C05437=1065.697,216.164,-85.426,173.240,30.452,155.567
C05438=1065.691,215.915,-85.400,173.238,30.449,155.567
C05439=1065.685,215.666,-85.375,173.236,30.444,155.566
C05440=1065.680,215.418,-85.348,173.234,30.440,155.565
C05441=1065.673,215.169,-85.323,173.232,30.436,155.564
C05442=1065.668,214.920,-85.297,173.230,30.432,155.564
C05443=1065.662,214.672,-85.272,173.228,30.428,155.563
C05444=1065.655,214.423,-85.246,173.225,30.424,155.562
C05445=1065.650,214.175,-85.220,173.224,30.420,155.561
C05446=1065.643,213.926,-85.194,173.222,30.416,155.561
C05447=1065.638,213.677,-85.168,173.219,30.411,155.560
C05448=1065.632,213.428,-85.143,173.218,30.408,155.559
C05449=1065.625,213.180,-85.117,173.216,30.403,155.559
C05450=1065.620,212.931,-85.091,173.214,30.399,155.558
C05451=1065.614,212.682,-85.066,173.212,30.395,155.557
C05452=1065.608,212.435,-85.041,173.210,30.391,155.556
C05453=1065.603,212.186,-85.015,173.208,30.387,155.556
C05454=1065.596,211.937,-84.989,173.206,30.383,155.555
C05455=1065.590,211.688,-84.964,173.204,30.379,155.554
C05456=1065.585,211.439,-84.938,173.202,30.375,155.554
C05457=1065.578,211.191,-84.913,173.200,30.371,155.553
C05458=1065.572,210.942,-84.887,173.198,30.367,155.552
C05459=1065.566,210.693,-84.862,173.196,30.363,155.552
C05460=1065.560,210.445,-84.837,173.194,30.359,155.551
C05461=1065.554,210.196,-84.811,173.192,30.355,155.550
C05462=1065.549,209.948,-84.786,173.190,30.350,155.549
C05463=1065.543,209.699,-84.761,173.188,30.347,155.549
C05464=1065.536,209.450,-84.735,173.186,30.342,155.548
C05465=1065.530,209.202,-84.710,173.184,30.338,155.547
C05466=1065.525,208.982,-84.687,173.182,30.335,155.547
C05467=1065.519,208.761,-84.665,173.180,30.331,155.546
C05468=1065.514,208.541,-84.642,173.179,30.327,155.545
C05469=1065.510,208.320,-84.619,173.177,30.324,155.545
C05470=1065.504,208.100,-84.597,173.175,30.320,155.544
C05471=1065.498,207.879,-84.575,173.174,30.316,155.543
C05472=1065.493,207.659,-84.553,173.172,30.313,155.543
C05473=1065.488,207.439,-84.531,173.170,30.309,155.542
C05474=1065.464,206.392,-84.427,173.012,30.231,155.537
C05475=1065.457,206.144,-84.402,173.011,30.228,155.536
C05476=1065.452,205.895,-84.378,173.008,30.225,155.536
C05477=1065.445,205.646,-84.354,173.006,30.221,155.535
C05478=1065.440,205.398,-84.329,173.004,30.219,155.535
C05479=1065.434,205.148,-84.305,173.001,30.215,155.534
C05480=1065.429,204.900,-84.280,172.999,30.212,155.534
C05481=1065.423,204.651,-84.255,172.997,30.209,155.533
C05482=1065.417,204.402,-84.231,172.995,30.205,155.533
C05483=1065.411,204.154,-84.207,172.992,30.202,155.532
C05484=1065.406,203.905,-84.183,172.990,30.199,155.532
C05485=1065.400,203.656,-84.158,172.988,30.196,155.531
C05486=1065.394,203.407,-84.134,172.986,30.193,155.531
C05487=1065.388,203.159,-84.110,172.983,30.189,155.530
C05488=1065.383,202.910,-84.086,172.982,30.186,155.530
C05489=1065.377,202.661,-84.060,172.979,30.183,155.529
C05490=1065.371,202.413,-84.036,172.977,30.180,155.529
C05491=1065.366,202.164,-84.011,172.975,30.177,155.528
C05492=1065.360,201.915,-83.988,172.973,30.174,155.528
C05493=1065.354,201.666,-83.963,172.970,30.171,155.527
C05494=1065.348,201.418,-83.940,172.969,30.167,155.527
C05495=1065.342,201.169,-83.915,172.966,30.165,155.526
C05496=1065.336,200.920,-83.891,172.964,30.161,155.526
C05497=1065.330,200.672,-83.867,172.961,30.158,155.525
C05498=1065.324,200.422,-83.844,172.960,30.155,155.525
C05499=1065.319,200.173,-83.819,172.957,30.152,155.524
C05500=1065.312,199.924,-83.795,172.955,30.149,155.524
C05501=1065.307,199.676,-83.771,172.953,30.146,155.523
C05502=1065.301,199.428,-83.747,172.951,30.143,155.523
C05503=1065.295,199.178,-83.723,172.948,30.140,155.522
C05504=1065.289,198.930,-83.699,172.947,30.137,155.522
C05505=1065.284,198.681,-83.675,172.944,30.133,155.521
C05506=1065.277,198.432,-83.651,172.942,30.131,155.521
C05507=1065.272,198.183,-83.627,172.939,30.127,155.520
C05508=1065.265,197.934,-83.603,172.938,30.125,155.520
C05509=1065.260,197.686,-83.579,172.935,30.121,155.519
C05510=1065.254,197.437,-83.555,172.933,30.118,155.519
C05511=1065.248,197.188,-83.531,172.932,30.115,155.519
C05512=1065.242,196.940,-83.507,172.929,30.112,155.518
C05513=1065.237,196.691,-83.484,172.927,30.109,155.518
C05514=1065.230,196.442,-83.460,172.925,30.106,155.517
C05515=1065.225,196.193,-83.435,172.923,30.103,155.517
C05516=1065.219,195.945,-83.412,172.920,30.100,155.516
C05517=1065.213,195.696,-83.389,172.919,30.097,155.516
C05518=1065.207,195.447,-83.364,172.916,30.094,155.515
C05519=1065.201,195.198,-83.340,172.914,30.090,155.515
C05520=1065.196,194.950,-83.316,172.911,30.087,155.514
C05521=1065.190,194.700,-83.293,172.910,30.084,155.514
C05522=1065.184,194.452,-83.269,172.908,30.081,155.513
C05523=1065.178,194.203,-83.245,172.905,30.078,155.513
C05524=1065.173,193.954,-83.221,172.904,30.075,155.512
C05525=1065.167,193.705,-83.197,172.901,30.072,155.512
C05526=1065.161,193.457,-83.174,172.899,30.069,155.511
C05527=1065.156,193.208,-83.150,172.897,30.066,155.511
C05528=1065.150,192.959,-83.127,172.895,30.063,155.510
C05529=1065.144,192.709,-83.103,172.893,30.060,155.510
C05530=1065.138,192.461,-83.079,172.891,30.056,155.509
C05531=1065.132,192.213,-83.055,172.889,30.054,155.509
C05532=1065.127,191.964,-83.032,172.886,30.050,155.508
C05533=1065.121,191.715,-83.008,172.884,30.048,155.508
C05534=1065.115,191.465,-82.984,172.883,30.044,155.507
C05535=1065.108,191.183,-82.957,172.880,30.041,155.507
C05536=1065.102,190.900,-82.930,172.877,30.038,155.506
C05537=1065.096,190.617,-82.904,172.875,30.034,155.506
C05538=1065.090,190.334,-82.877,172.873,30.030,155.505
C05539=1065.084,190.086,-82.853,172.870,30.027,155.505
C05540=1065.078,189.837,-82.830,172.869,30.024,155.504
C05541=1065.073,189.588,-82.806,172.866,30.021,155.504
C05542=1065.067,189.340,-82.783,172.864,30.018,155.503
C05543=1065.061,189.091,-82.759,172.863,30.015,155.503
C05544=1065.055,188.841,-82.735,172.860,30.012,155.503
C05545=1065.049,188.592,-82.712,172.858,30.009,155.502
C05546=1065.044,188.344,-82.688,172.857,30.006,155.502
C05547=1065.038,188.095,-82.665,172.854,30.003,155.501
C05548=1065.032,187.847,-82.642,172.852,30.000,155.501
C05549=1065.027,187.598,-82.618,172.850,29.997,155.500
C05550=1065.022,187.349,-82.595,172.848,29.993,155.500
C05551=1065.016,187.100,-82.571,172.846,29.991,155.499
C05552=1065.011,186.851,-82.548,172.844,29.987,155.499
C05553=1065.005,186.603,-82.524,172.842,29.985,155.498
C05554=1064.998,186.353,-82.501,172.840,29.981,155.498
C05555=1064.993,186.104,-82.477,172.837,29.978,155.497
C05556=1064.987,185.856,-82.454,172.836,29.975,155.497
C05557=1064.981,185.607,-82.431,172.834,29.972,155.496
C05558=1064.976,185.358,-82.407,172.831,29.969,155.496
C05559=1064.971,185.109,-82.384,172.830,29.966,155.495
C05560=1064.965,184.861,-82.361,172.828,29.963,155.495
C05561=1064.960,184.611,-82.337,172.825,29.960,155.494
C05562=1064.954,184.362,-82.314,172.824,29.957,155.494
C05563=1064.948,184.113,-82.291,172.822,29.954,155.493
C05564=1064.942,183.865,-82.269,172.819,29.951,155.493
C05565=1064.935,183.616,-82.245,172.818,29.949,155.493
C05566=1064.929,183.367,-82.222,172.815,29.945,155.492
C05567=1064.924,183.118,-82.199,172.813,29.942,155.492
C05568=1064.918,182.869,-82.176,172.811,29.940,155.491
C05569=1064.912,182.620,-82.153,172.809,29.937,155.491
C05570=1064.906,182.371,-82.130,172.807,29.934,155.490
C05571=1064.900,182.123,-82.106,172.805,29.931,155.490
C05572=1064.893,181.874,-82.084,172.803,29.928,155.490
C05573=1064.888,181.625,-82.061,172.801,29.925,155.489
C05574=1064.882,181.376,-82.038,172.799,29.922,155.489
C05575=1064.876,181.127,-82.015,172.797,29.919,155.488
C05576=1064.870,180.878,-81.992,172.795,29.916,155.488
C05577=1064.865,180.629,-81.969,172.793,29.914,155.487
C05578=1064.859,180.381,-81.946,172.790,29.911,155.487
C05579=1064.853,180.132,-81.924,172.789,29.908,155.486
C05580=1064.847,179.883,-81.901,172.787,29.905,155.486
C05581=1064.841,179.634,-81.878,172.784,29.902,155.486
C05582=1064.835,179.385,-81.855,172.783,29.899,155.485
C05583=1064.830,179.136,-81.832,172.781,29.896,155.485
C05584=1064.824,178.887,-81.809,172.778,29.893,155.484
C05585=1064.817,178.639,-81.787,172.777,29.890,155.484
C05586=1064.812,178.390,-81.764,172.775,29.887,155.483
C05587=1064.805,178.140,-81.740,172.772,29.884,155.483
C05588=1064.800,177.891,-81.717,172.771,29.882,155.482
C05589=1064.794,177.643,-81.694,172.769,29.879,155.482
C05590=1064.788,177.394,-81.671,172.767,29.876,155.482
C05591=1064.782,177.145,-81.649,172.764,29.873,155.481
C05592=1064.776,176.896,-81.626,172.763,29.870,155.481
C05593=1064.770,176.647,-81.603,172.761,29.867,155.480
C05594=1064.765,176.398,-81.581,172.758,29.864,155.480
C05595=1064.759,176.149,-81.558,172.757,29.861,155.479
C05596=1064.753,175.901,-81.536,172.755,29.858,155.479
C05597=1064.747,175.652,-81.513,172.753,29.855,155.478
C05598=1064.742,175.403,-81.490,172.751,29.853,155.478
C05599=1064.735,175.120,-81.464,172.749,29.849,155.478
C05600=1064.729,174.836,-81.439,172.746,29.846,155.477
C05601=1064.722,174.553,-81.413,172.744,29.842,155.477
C05602=1064.716,174.270,-81.387,172.742,29.839,155.476
C05603=1064.709,174.022,-81.364,172.740,29.837,155.476
C05604=1064.704,173.772,-81.342,172.738,29.834,155.475
C05605=1064.698,173.523,-81.319,172.736,29.830,155.475
C05606=1064.692,173.274,-81.296,172.734,29.828,155.474
C05607=1064.686,173.026,-81.274,172.733,29.825,155.474
C05608=1064.680,172.776,-81.252,172.730,29.822,155.473
C05609=1064.675,172.527,-81.229,172.728,29.819,155.473
C05610=1064.669,172.278,-81.206,172.727,29.816,155.472
C05611=1064.662,172.030,-81.183,172.725,29.813,155.472
C05612=1064.658,171.781,-81.162,172.722,29.810,155.472
C05613=1064.652,171.532,-81.139,172.720,29.807,155.471
C05614=1064.646,171.283,-81.116,172.719,29.805,155.471
C05615=1064.640,171.034,-81.094,172.717,29.802,155.470
C05616=1064.634,170.785,-81.071,172.714,29.799,155.470
C05617=1064.629,170.536,-81.048,172.713,29.796,155.469
C05618=1064.623,170.287,-81.026,172.711,29.793,155.469
C05619=1064.617,170.039,-81.004,172.709,29.790,155.468
C05620=1064.612,169.790,-80.981,172.707,29.787,155.468
C05621=1064.606,169.540,-80.959,172.705,29.784,155.468
C05622=1064.600,169.292,-80.936,172.703,29.781,155.467
C05623=1064.594,169.042,-80.914,172.702,29.779,155.467
C05624=1064.589,168.794,-80.892,172.699,29.775,155.466
C05625=1064.583,168.545,-80.869,172.697,29.772,155.466
C05626=1064.577,168.296,-80.847,172.696,29.770,155.465
C05627=1064.571,168.047,-80.824,172.694,29.767,155.465
C05628=1064.566,167.798,-80.802,172.692,29.764,155.464
C05629=1064.560,167.550,-80.780,172.690,29.761,155.464
C05630=1064.555,167.300,-80.758,172.688,29.758,155.464
C05631=1064.549,167.051,-80.735,172.686,29.755,155.463
C05632=1064.543,166.802,-80.713,172.684,29.752,155.463
C05633=1064.538,166.554,-80.691,172.682,29.749,155.462
C05634=1064.532,166.304,-80.668,172.680,29.746,155.462
C05635=1064.527,166.055,-80.645,172.678,29.744,155.461
C05636=1064.520,165.806,-80.624,172.677,29.740,155.461
C05637=1064.515,165.558,-80.601,172.675,29.738,155.460
C05638=1064.510,165.308,-80.579,172.672,29.735,155.460
C05639=1064.503,165.060,-80.557,172.671,29.731,155.459
C05640=1064.498,164.810,-80.534,172.669,29.729,155.459
C05641=1064.493,164.562,-80.512,172.667,29.726,155.459
C05642=1064.487,164.313,-80.490,172.666,29.723,155.458
C05643=1064.481,164.063,-80.468,172.664,29.720,155.458
C05644=1064.476,163.815,-80.445,172.661,29.717,155.457
C05645=1064.470,163.566,-80.424,172.660,29.714,155.457
C05646=1064.465,163.317,-80.401,172.658,29.711,155.456
C05647=1064.459,163.068,-80.379,172.656,29.709,155.456
C05648=1064.453,162.819,-80.357,172.655,29.705,155.455
C05649=1064.448,162.570,-80.335,172.652,29.702,155.455
C05650=1064.442,162.322,-80.313,172.650,29.699,155.455
C05651=1064.437,162.072,-80.291,172.649,29.697,155.454
C05652=1064.431,161.823,-80.269,172.647,29.694,155.454
C05653=1064.425,161.575,-80.247,172.645,29.691,155.453
C05654=1064.420,161.325,-80.224,172.644,29.688,155.453
C05655=1064.414,161.076,-80.202,172.641,29.685,155.452
C05656=1064.409,160.827,-80.181,172.639,29.682,155.452
C05657=1064.402,160.579,-80.158,172.638,29.679,155.451
C05658=1064.396,160.329,-80.137,172.636,29.676,155.451
C05659=1064.391,160.081,-80.115,172.634,29.674,155.451
C05660=1064.385,159.831,-80.093,172.632,29.671,155.450
C05661=1064.379,159.583,-80.071,172.630,29.668,155.450
C05662=1064.373,159.333,-80.049,172.628,29.665,155.449
C05663=1064.366,159.050,-80.024,172.626,29.662,155.449
C05664=1064.361,158.766,-80.000,172.624,29.659,155.448
C05665=1064.354,158.483,-79.975,172.622,29.655,155.448
C05666=1064.347,158.199,-79.950,172.620,29.653,155.447
C05667=1064.341,157.950,-79.928,172.618,29.649,155.447
C05668=1064.335,157.701,-79.906,172.616,29.647,155.447
C05669=1064.330,157.452,-79.885,172.615,29.644,155.446
C05670=1064.324,157.203,-79.862,172.613,29.641,155.446
C05671=1064.318,156.954,-79.841,172.611,29.638,155.445
C05672=1064.312,156.706,-79.819,172.608,29.636,155.445
C05673=1064.306,156.456,-79.798,172.607,29.632,155.444
C05674=1064.301,156.207,-79.776,172.605,29.630,155.444
C05675=1064.295,155.958,-79.754,172.603,29.627,155.444
C05676=1064.289,155.709,-79.733,172.602,29.624,155.443
C05677=1064.283,155.461,-79.711,172.600,29.622,155.443
C05678=1064.278,155.211,-79.689,172.598,29.618,155.442
C05679=1064.272,154.962,-79.667,172.597,29.616,155.442
C05680=1064.266,154.713,-79.646,172.594,29.613,155.441
C05681=1064.260,154.464,-79.625,172.592,29.610,155.441
C05682=1064.254,154.215,-79.603,172.591,29.607,155.441
C05683=1064.248,153.967,-79.582,172.589,29.605,155.440
C05684=1064.243,153.717,-79.559,172.587,29.602,155.440
C05685=1064.237,153.469,-79.538,172.586,29.599,155.439
C05686=1064.231,153.219,-79.517,172.584,29.596,155.439
C05687=1064.225,152.970,-79.495,172.581,29.593,155.438
C05688=1064.219,152.722,-79.474,172.580,29.590,155.438
C05689=1064.213,152.472,-79.452,172.578,29.588,155.438
C05690=1064.208,152.224,-79.431,172.576,29.585,155.437
C05691=1064.203,151.974,-79.409,172.575,29.582,155.437
C05692=1064.197,151.725,-79.388,172.573,29.580,155.436
C05693=1064.191,151.476,-79.366,172.571,29.576,155.436
C05694=1064.185,151.227,-79.345,172.570,29.574,155.435
C05695=1064.179,150.978,-79.323,172.568,29.571,155.435
C05696=1064.173,150.729,-79.302,172.565,29.568,155.435
C05697=1064.167,150.481,-79.280,172.563,29.565,155.434
C05698=1064.162,150.231,-79.260,172.562,29.563,155.434
C05699=1064.156,149.982,-79.238,172.560,29.560,155.433
C05700=1064.150,149.733,-79.217,172.558,29.557,155.433
C05701=1064.144,149.485,-79.195,172.557,29.554,155.432
C05702=1064.139,149.235,-79.173,172.555,29.551,155.432
C05703=1064.134,148.986,-79.153,172.553,29.548,155.432
C05704=1064.127,148.737,-79.131,172.552,29.546,155.431
C05705=1064.121,148.488,-79.109,172.550,29.543,155.431
C05706=1064.116,148.239,-79.088,172.547,29.540,155.430
C05707=1064.110,147.989,-79.067,172.546,29.537,155.430
C05708=1064.104,147.741,-79.046,172.544,29.534,155.430
C05709=1064.098,147.491,-79.024,172.542,29.531,155.429
C05710=1064.092,147.243,-79.004,172.541,29.529,155.429
C05711=1064.086,146.993,-78.983,172.539,29.526,155.428
C05712=1064.080,146.745,-78.961,172.537,29.523,155.428
C05713=1064.074,146.496,-78.940,172.536,29.521,155.427
C05714=1064.069,146.247,-78.919,172.534,29.518,155.427
C05715=1064.063,145.997,-78.898,172.532,29.515,155.427
C05716=1064.057,145.749,-78.876,172.531,29.513,155.426
C05717=1064.051,145.499,-78.855,172.528,29.510,155.426
C05718=1064.046,145.251,-78.834,172.526,29.507,155.425
C05719=1064.039,145.002,-78.813,172.525,29.504,155.425
C05720=1064.034,144.753,-78.793,172.523,29.502,155.425
C05721=1064.028,144.503,-78.771,172.521,29.498,155.424
C05722=1064.022,144.254,-78.750,172.520,29.496,155.424
C05723=1064.016,144.005,-78.729,172.518,29.493,155.423
C05724=1064.011,143.757,-78.707,172.516,29.490,155.423
C05725=1064.005,143.507,-78.687,172.515,29.487,155.422
C05726=1063.998,143.259,-78.666,172.513,29.485,155.422
C05727=1063.990,142.870,-78.633,172.510,29.481,155.421
C05728=1063.981,142.481,-78.600,172.507,29.476,155.421
C05729=1063.972,142.093,-78.567,172.504,29.472,155.420
C05730=1063.963,141.704,-78.535,172.502,29.467,155.419
C05731=1063.957,141.454,-78.514,172.500,29.464,155.419
C05732=1063.951,141.206,-78.493,172.499,29.462,155.419
C05733=1063.946,140.956,-78.472,172.497,29.459,155.418
C05734=1063.940,140.707,-78.451,172.495,29.456,155.418
C05735=1063.931,140.314,-78.418,172.492,29.452,155.417
C05736=1063.921,139.920,-78.385,172.489,29.447,155.416
C05737=1063.912,139.528,-78.352,172.487,29.443,155.416
C05738=1063.903,139.134,-78.319,172.484,29.439,155.415
C05739=1063.898,138.885,-78.298,172.483,29.436,155.415
C05740=1063.891,138.636,-78.278,172.481,29.433,155.414
C05741=1063.886,138.387,-78.257,172.479,29.431,155.414
C05742=1063.880,138.137,-78.236,172.478,29.428,155.413
C05743=1063.874,137.889,-78.216,172.476,29.425,155.413
C05744=1063.868,137.639,-78.195,172.474,29.422,155.413
C05745=1063.862,137.390,-78.173,172.472,29.419,155.412
C05746=1063.856,137.141,-78.153,172.470,29.417,155.412
C05747=1063.851,136.892,-78.133,172.468,29.414,155.411
C05748=1063.844,136.643,-78.112,172.467,29.411,155.411
C05749=1063.839,136.394,-78.091,172.465,29.409,155.411
C05750=1063.833,136.144,-78.070,172.463,29.406,155.410
C05751=1063.827,135.896,-78.050,172.462,29.403,155.410
C05752=1063.821,135.647,-78.029,172.460,29.401,155.409
C05753=1063.815,135.398,-78.009,172.458,29.398,155.409
C05754=1063.809,135.149,-77.988,172.456,29.395,155.409
C05755=1063.804,134.900,-77.967,172.455,29.392,155.408
C05756=1063.797,134.650,-77.947,172.453,29.390,155.408
C05757=1063.792,134.401,-77.926,172.452,29.386,155.407
C05758=1063.786,134.153,-77.906,172.450,29.384,155.407
C05759=1063.780,133.903,-77.885,172.448,29.381,155.406
C05760=1063.775,133.654,-77.864,172.447,29.378,155.406
C05761=1063.769,133.405,-77.844,172.445,29.375,155.406
C05762=1063.763,133.156,-77.823,172.443,29.373,155.405
C05763=1063.757,132.907,-77.803,172.441,29.370,155.405
C05764=1063.752,132.658,-77.783,172.440,29.367,155.404
C05765=1063.746,132.409,-77.761,172.438,29.365,155.404
C05766=1063.739,132.160,-77.741,172.436,29.362,155.404
C05767=1063.734,131.911,-77.720,172.435,29.359,155.403
C05768=1063.728,131.662,-77.700,172.433,29.356,155.403
C05769=1063.722,131.412,-77.680,172.431,29.354,155.402
C05770=1063.716,131.163,-77.660,172.430,29.351,155.402
C05771=1063.710,130.914,-77.640,172.428,29.348,155.402
C05772=1063.704,130.665,-77.619,172.426,29.346,155.401
C05773=1063.698,130.416,-77.599,172.425,29.343,155.401
C05774=1063.692,130.167,-77.579,172.423,29.340,155.400
C05775=1063.686,129.918,-77.559,172.421,29.337,155.400
C05776=1063.681,129.668,-77.538,172.420,29.335,155.400
C05777=1063.675,129.419,-77.518,172.418,29.332,155.399
C05778=1063.668,129.171,-77.497,172.416,29.329,155.399
C05779=1063.662,128.921,-77.476,172.415,29.327,155.398
C05780=1063.656,128.673,-77.456,172.413,29.324,155.398
C05781=1063.650,128.424,-77.436,172.411,29.322,155.398
C05782=1063.645,128.174,-77.417,172.410,29.319,155.397
C05783=1063.639,127.924,-77.396,172.408,29.316,155.397
C05784=1063.633,127.676,-77.376,172.406,29.314,155.396
C05785=1063.627,127.427,-77.356,172.405,29.311,155.396
C05786=1063.621,127.177,-77.335,172.403,29.308,155.396
C05787=1063.614,126.894,-77.312,172.401,29.305,155.395
C05788=1063.607,126.610,-77.290,172.399,29.302,155.395
C05789=1063.601,126.326,-77.267,172.397,29.299,155.394
C05790=1063.594,126.042,-77.243,172.396,29.296,155.394
C05791=1063.589,125.792,-77.224,172.394,29.293,155.393
C05792=1063.583,125.543,-77.204,172.392,29.290,155.393
C05793=1063.576,125.294,-77.183,172.391,29.288,155.393
C05794=1063.570,125.045,-77.163,172.389,29.285,155.392
C05795=1063.565,124.796,-77.143,172.387,29.282,155.392
C05796=1063.559,124.547,-77.123,172.386,29.279,155.391
C05797=1063.553,124.298,-77.103,172.384,29.277,155.391
C05798=1063.546,124.049,-77.082,172.382,29.274,155.391
C05799=1063.541,123.799,-77.063,172.381,29.271,155.390
C05800=1063.535,123.550,-77.043,172.379,29.269,155.390
C05801=1063.529,123.301,-77.023,172.377,29.266,155.389
C05802=1063.523,123.053,-77.003,172.376,29.263,155.389
C05803=1063.518,122.803,-76.982,172.374,29.260,155.388
C05804=1063.512,122.553,-76.963,172.372,29.258,155.388
C05805=1063.506,122.304,-76.943,172.371,29.255,155.388
C05806=1063.500,122.056,-76.923,172.369,29.252,155.387
C05807=1063.495,121.807,-76.902,172.367,29.250,155.387
C05808=1063.489,121.557,-76.883,172.366,29.247,155.386
C05809=1063.483,121.308,-76.863,172.365,29.244,155.386
C05810=1063.476,121.059,-76.843,172.363,29.242,155.386
C05811=1063.470,120.810,-76.823,172.362,29.239,155.385
C05812=1063.465,120.560,-76.803,172.360,29.236,155.385
C05813=1063.459,120.311,-76.783,172.358,29.233,155.384
C05814=1063.453,120.063,-76.763,172.357,29.231,155.384
C05815=1063.447,119.814,-76.743,172.355,29.228,155.384
C05816=1063.443,119.564,-76.723,172.353,29.225,155.383
C05817=1063.437,119.315,-76.703,172.352,29.222,155.383
C05818=1063.431,119.066,-76.683,172.350,29.219,155.382
C05819=1063.425,118.817,-76.664,172.348,29.216,155.382
C05820=1063.418,118.567,-76.644,172.347,29.214,155.381
C05821=1063.413,118.318,-76.623,172.345,29.211,155.381
C05822=1063.407,118.069,-76.604,172.343,29.208,155.381
C05823=1063.401,117.820,-76.584,172.342,29.205,155.380
C05824=1063.396,117.571,-76.565,172.340,29.203,155.380
C05825=1063.390,117.322,-76.545,172.338,29.200,155.379
C05826=1063.384,117.073,-76.524,172.337,29.197,155.379
C05827=1063.379,116.823,-76.505,172.335,29.195,155.379
C05828=1063.373,116.574,-76.485,172.334,29.192,155.378
C05829=1063.367,116.325,-76.466,172.333,29.189,155.378
C05830=1063.361,116.076,-76.446,172.331,29.187,155.377
C05831=1063.355,115.827,-76.426,172.329,29.184,155.377
C05832=1063.350,115.578,-76.406,172.328,29.181,155.377
C05833=1063.344,115.329,-76.386,172.326,29.178,155.376
C05834=1063.338,115.079,-76.367,172.325,29.175,155.376
C05835=1063.332,114.831,-76.347,172.323,29.172,155.375
C05836=1063.327,114.581,-76.327,172.321,29.170,155.375
C05837=1063.321,114.332,-76.308,172.320,29.167,155.374
C05838=1063.316,114.083,-76.288,172.318,29.164,155.374
C05839=1063.309,113.834,-76.268,172.316,29.161,155.374
C05840=1063.303,113.585,-76.249,172.315,29.159,155.373
C05841=1063.297,113.336,-76.229,172.313,29.156,155.373
C05842=1063.292,113.086,-76.210,172.312,29.153,155.372
C05843=1063.286,112.838,-76.190,172.311,29.151,155.372
C05844=1063.280,112.588,-76.171,172.309,29.148,155.372
C05845=1063.274,112.339,-76.151,172.307,29.145,155.371
C05846=1063.268,112.090,-76.131,172.306,29.142,155.371
C05847=1063.263,111.841,-76.112,172.304,29.140,155.370
C05848=1063.257,111.592,-76.092,172.302,29.137,155.370
C05849=1063.251,111.342,-76.073,172.301,29.134,155.370
C05850=1063.245,111.093,-76.054,172.299,29.132,155.369
C05851=1063.238,110.808,-76.031,172.297,29.129,155.369
C05852=1063.232,110.525,-76.009,172.296,29.126,155.368
C05853=1063.224,110.240,-75.987,172.294,29.123,155.368
C05854=1063.217,109.957,-75.965,172.292,29.120,155.367
C05855=1063.212,109.707,-75.946,172.290,29.117,155.367
C05856=1063.206,109.458,-75.926,172.289,29.115,155.367
C05857=1063.200,109.209,-75.907,172.288,29.112,155.366
C05858=1063.194,108.960,-75.888,172.286,29.109,155.366
C05859=1063.188,108.710,-75.869,172.284,29.106,155.365
C05860=1063.182,108.461,-75.849,172.283,29.104,155.365
C05861=1063.176,108.212,-75.830,172.281,29.101,155.365
C05862=1063.171,107.963,-75.810,172.279,29.098,155.364
C05863=1063.164,107.714,-75.791,172.278,29.095,155.364
C05864=1063.158,107.465,-75.772,172.276,29.093,155.363
C05865=1063.152,107.215,-75.752,172.274,29.090,155.363
C05866=1063.147,106.966,-75.733,172.273,29.087,155.363
C05867=1063.140,106.717,-75.715,172.271,29.084,155.362
C05868=1063.134,106.468,-75.695,172.270,29.082,155.362
C05869=1063.129,106.218,-75.675,172.269,29.079,155.361
C05870=1063.123,105.969,-75.656,172.267,29.077,155.361
C05871=1063.117,105.720,-75.637,172.265,29.074,155.361
C05872=1063.111,105.471,-75.619,172.264,29.071,155.360
C05873=1063.105,105.222,-75.599,172.262,29.069,155.360
C05874=1063.100,104.973,-75.579,172.260,29.066,155.359
C05875=1063.094,104.723,-75.560,172.259,29.063,155.359
C05876=1063.088,104.474,-75.541,172.257,29.061,155.359
C05877=1063.082,104.225,-75.522,172.256,29.058,155.358
C05878=1063.076,103.975,-75.503,172.255,29.055,155.358
C05879=1063.070,103.727,-75.483,172.253,29.053,155.357
C05880=1063.064,103.478,-75.464,172.252,29.050,155.357
C05881=1063.058,103.228,-75.445,172.250,29.047,155.357
C05882=1063.053,102.979,-75.426,172.248,29.044,155.356
C05883=1063.047,102.730,-75.408,172.247,29.042,155.356
C05884=1063.041,102.481,-75.388,172.245,29.039,155.355
C05885=1063.035,102.231,-75.369,172.243,29.036,155.355
C05886=1063.030,101.982,-75.350,172.242,29.033,155.355
C05887=1063.023,101.733,-75.331,172.241,29.031,155.354
C05888=1063.017,101.483,-75.312,172.239,29.028,155.354
C05889=1063.012,101.235,-75.293,172.238,29.025,155.353
C05890=1063.007,100.985,-75.274,172.236,29.023,155.353
C05891=1063.000,100.736,-75.255,172.234,29.020,155.353
C05892=1062.995,100.487,-75.236,172.233,29.017,155.352
C05893=1062.988,100.238,-75.217,172.231,29.014,155.352
C05894=1062.982,99.988,-75.198,172.230,29.012,155.351
C05895=1062.976,99.739,-75.179,172.228,29.009,155.351
C05896=1062.970,99.490,-75.160,172.227,29.006,155.350
C05897=1062.964,99.240,-75.142,172.226,29.004,155.350
C05898=1062.959,98.992,-75.123,172.224,29.001,155.350
C05899=1062.952,98.743,-75.104,172.222,28.999,155.349
C05900=1062.947,98.493,-75.085,172.221,28.996,155.349
C05901=1062.940,98.244,-75.066,172.219,28.993,155.349
C05902=1062.935,97.995,-75.047,172.217,28.990,155.348
C05903=1062.928,97.745,-75.028,172.216,28.988,155.348
C05904=1062.923,97.496,-75.009,172.214,28.985,155.347
C05905=1062.917,97.248,-74.991,172.213,28.982,155.347
C05906=1062.911,96.998,-74.971,172.212,28.980,155.347
C05907=1062.905,96.748,-74.954,172.210,28.977,155.346
C05908=1062.899,96.499,-74.934,172.208,28.975,155.346
C05909=1062.893,96.250,-74.916,172.207,28.972,155.345
C05910=1062.888,96.001,-74.897,172.205,28.969,155.345
C05911=1062.881,95.752,-74.878,172.204,28.966,155.345
C05912=1062.875,95.503,-74.859,172.202,28.964,155.344
C05913=1062.869,95.254,-74.840,172.201,28.961,155.344
C05914=1062.863,95.004,-74.822,172.200,28.958,155.343
C05915=1062.857,94.719,-74.801,172.198,28.955,155.343
C05916=1062.850,94.436,-74.780,172.195,28.952,155.343
C05917=1062.843,94.152,-74.757,172.194,28.949,155.342
C05918=1062.836,93.868,-74.736,172.192,28.946,155.342
C05919=1062.830,93.618,-74.718,172.191,28.943,155.341
C05920=1062.825,93.369,-74.700,172.189,28.940,155.341
C05921=1062.819,93.120,-74.681,172.188,28.938,155.340
C05922=1062.813,92.871,-74.662,172.187,28.935,155.340
C05923=1062.807,92.621,-74.644,172.185,28.932,155.340
C05924=1062.802,92.372,-74.625,172.183,28.930,155.339
C05925=1062.795,92.123,-74.606,172.182,28.927,155.339
C05926=1062.790,91.874,-74.587,172.180,28.924,155.338
C05927=1062.784,91.625,-74.569,172.178,28.921,155.338
C05928=1062.778,91.376,-74.551,172.178,28.919,155.338
C05929=1062.772,91.126,-74.531,172.176,28.916,155.337
C05930=1062.766,90.876,-74.514,172.175,28.913,155.337
C05931=1062.761,90.628,-74.495,172.173,28.911,155.336
C05932=1062.754,90.379,-74.476,172.171,28.908,155.336
C05933=1062.748,90.129,-74.458,172.170,28.906,155.336
C05934=1062.742,89.880,-74.439,172.168,28.903,155.335
C05935=1062.736,89.631,-74.421,172.166,28.900,155.335
C05936=1062.731,89.381,-74.403,172.166,28.898,155.334
C05937=1062.724,89.132,-74.384,172.164,28.895,155.334
C05938=1062.718,88.882,-74.366,172.162,28.892,155.334
C05939=1062.712,88.634,-74.348,172.161,28.890,155.333
C05940=1062.707,88.385,-74.328,172.159,28.887,155.333
C05941=1062.700,88.135,-74.311,172.157,28.884,155.333
C05942=1062.694,87.886,-74.292,172.156,28.882,155.332
C05943=1062.688,87.637,-74.274,172.155,28.879,155.332
C05944=1062.682,87.388,-74.256,172.154,28.876,155.331
C05945=1062.676,87.138,-74.238,172.152,28.874,155.331
C05946=1062.671,86.889,-74.219,172.150,28.871,155.331
C05947=1062.664,86.640,-74.200,172.149,28.869,155.330
C05948=1062.658,86.390,-74.182,172.147,28.866,155.330
C05949=1062.652,86.141,-74.164,172.145,28.863,155.329
C05950=1062.646,85.892,-74.146,172.145,28.861,155.329
C05951=1062.641,85.643,-74.127,172.143,28.858,155.329
C05952=1062.635,85.393,-74.109,172.141,28.855,155.328
C05953=1062.629,85.144,-74.091,172.140,28.852,155.328
C05954=1062.623,84.895,-74.073,172.138,28.850,155.327
C05955=1062.616,84.646,-74.054,172.136,28.847,155.327
C05956=1062.611,84.397,-74.036,172.135,28.845,155.327
C05957=1062.605,84.147,-74.019,172.134,28.842,155.326
C05958=1062.599,83.897,-73.999,172.133,28.839,155.326
C05959=1062.593,83.648,-73.982,172.131,28.837,155.326
C05960=1062.587,83.399,-73.963,172.129,28.834,155.325
C05961=1062.581,83.150,-73.946,172.128,28.831,155.325
C05962=1062.575,82.901,-73.927,172.126,28.828,155.324
C05963=1062.569,82.651,-73.909,172.124,28.826,155.324
C05964=1062.564,82.402,-73.891,172.124,28.823,155.323
C05965=1062.558,82.153,-73.872,172.122,28.820,155.323
C05966=1062.552,81.903,-73.854,172.120,28.818,155.323
C05967=1062.546,81.655,-73.836,172.119,28.815,155.322
C05968=1062.540,81.405,-73.818,172.117,28.813,155.322
C05969=1062.534,81.156,-73.800,172.116,28.810,155.322
C05970=1062.528,80.907,-73.782,172.115,28.807,155.321
C05971=1062.522,80.658,-73.764,172.113,28.804,155.321
C05972=1062.517,80.408,-73.746,172.112,28.802,155.320
C05973=1062.510,80.159,-73.727,172.110,28.799,155.320
C05974=1062.505,79.910,-73.709,172.108,28.796,155.320
C05975=1062.499,79.660,-73.692,172.107,28.793,155.319
C05976=1062.493,79.411,-73.673,172.105,28.791,155.319
C05977=1062.487,79.162,-73.655,172.105,28.788,155.318
C05978=1062.481,78.913,-73.638,172.103,28.785,155.318
C05979=1062.474,78.629,-73.617,172.101,28.783,155.318
C05980=1062.468,78.344,-73.596,172.100,28.779,155.317
C05981=1062.461,78.059,-73.576,172.098,28.776,155.317
C05982=1062.454,77.775,-73.555,172.096,28.774,155.316
C05983=1062.448,77.526,-73.538,172.095,28.771,155.316
C05984=1062.442,77.277,-73.520,172.093,28.768,155.315
C05985=1062.436,77.029,-73.502,172.092,28.765,155.315
C05986=1062.430,76.779,-73.484,172.090,28.763,155.315
C05987=1062.424,76.530,-73.466,172.088,28.760,155.314
C05988=1062.418,76.280,-73.448,172.087,28.758,155.314
C05989=1062.412,76.030,-73.431,172.086,28.755,155.314
C05990=1062.406,75.782,-73.412,172.084,28.752,155.313
C05991=1062.400,75.532,-73.394,172.083,28.750,155.313
C05992=1062.394,75.283,-73.377,172.081,28.747,155.312
C05993=1062.388,75.033,-73.359,172.080,28.744,155.312
C05994=1062.382,74.785,-73.342,172.078,28.741,155.312
C05995=1062.376,74.535,-73.324,172.076,28.739,155.311
C05996=1062.370,74.286,-73.306,172.076,28.737,155.311
C05997=1062.364,74.036,-73.288,172.074,28.734,155.310
C05998=1062.358,73.788,-73.270,172.072,28.731,155.310
C05999=1062.352,73.538,-73.252,172.071,28.728,155.310
C06000=1062.347,73.289,-73.235,172.069,28.726,155.309
C06001=1062.341,73.039,-73.217,172.068,28.723,155.309
C06002=1062.334,72.790,-73.200,172.067,28.721,155.309
C06003=1062.328,72.541,-73.182,172.065,28.718,155.308
C06004=1062.323,72.292,-73.164,172.064,28.715,155.308
C06005=1062.317,72.042,-73.146,172.062,28.712,155.307
C06006=1062.311,71.793,-73.129,172.060,28.710,155.307
C06007=1062.305,71.543,-73.111,172.059,28.707,155.307
C06008=1062.299,71.294,-73.094,172.058,28.704,155.306
C06009=1062.293,71.045,-73.076,172.057,28.702,155.306
C06010=1062.287,70.796,-73.058,172.055,28.699,155.305
C06011=1062.281,70.546,-73.040,172.053,28.697,155.305
C06012=1062.275,70.297,-73.023,172.052,28.694,155.305
C06013=1062.269,70.047,-73.006,172.050,28.691,155.304
C06014=1062.263,69.798,-72.988,172.049,28.689,155.304
C06015=1062.257,69.549,-72.970,172.048,28.686,155.303
C06016=1062.251,69.300,-72.952,172.046,28.683,155.303
C06017=1062.245,69.050,-72.935,172.044,28.681,155.303
C06018=1062.239,68.801,-72.918,172.043,28.678,155.302
C06019=1062.233,68.551,-72.900,172.041,28.675,155.302
C06020=1062.227,68.303,-72.883,172.041,28.673,155.301
C06021=1062.221,68.054,-72.865,172.039,28.670,155.301
C06022=1062.215,67.804,-72.847,172.037,28.667,155.301
C06023=1062.210,67.555,-72.830,172.036,28.665,155.300
C06024=1062.203,67.305,-72.813,172.034,28.662,155.300
C06025=1062.197,67.056,-72.795,172.032,28.659,155.300
C06026=1062.191,66.806,-72.777,172.032,28.657,155.299
C06027=1062.185,66.557,-72.760,172.030,28.654,155.299
C06028=1062.179,66.308,-72.743,172.029,28.652,155.299
C06029=1062.173,66.059,-72.726,172.027,28.649,155.298
C06030=1062.167,65.810,-72.708,172.025,28.646,155.298
C06031=1062.161,65.559,-72.691,172.024,28.644,155.297
C06032=1062.155,65.311,-72.674,172.023,28.641,155.297
C06033=1062.149,65.061,-72.656,172.021,28.638,155.297
C06034=1062.143,64.812,-72.638,172.020,28.636,155.296
C06035=1062.137,64.563,-72.621,172.018,28.633,155.296
C06036=1062.131,64.313,-72.603,172.017,28.630,155.295
C06037=1062.125,64.064,-72.587,172.015,28.628,155.295
C06038=1062.119,63.814,-72.569,172.014,28.626,155.295
C06039=1062.113,63.566,-72.552,172.013,28.623,155.294
C06040=1062.107,63.316,-72.534,172.011,28.620,155.294
C06041=1062.101,63.067,-72.518,172.009,28.617,155.294
C06042=1062.094,62.817,-72.501,172.008,28.615,155.293
C06043=1062.088,62.533,-72.481,172.006,28.612,155.293
C06044=1062.080,62.249,-72.461,172.005,28.609,155.292
C06045=1062.073,61.964,-72.442,172.003,28.606,155.292
C06046=1062.066,61.680,-72.423,172.001,28.604,155.292
C06047=1062.060,61.431,-72.405,172.000,28.601,155.291
C06048=1062.054,61.182,-72.388,171.998,28.598,155.291
C06049=1062.048,60.933,-72.372,171.996,28.596,155.290
C06050=1062.042,60.683,-72.354,171.996,28.593,155.290
C06051=1062.036,60.434,-72.337,171.994,28.590,155.290
C06052=1062.030,60.184,-72.319,171.993,28.588,155.289
C06053=1062.024,59.935,-72.302,171.991,28.585,155.289
C06054=1062.018,59.686,-72.286,171.989,28.583,155.289
C06055=1062.012,59.436,-72.268,171.988,28.580,155.288
C06056=1062.005,59.187,-72.251,171.987,28.578,155.288
C06057=1062.000,58.937,-72.234,171.985,28.575,155.287
C06058=1061.993,58.688,-72.217,171.984,28.572,155.287
C06059=1061.987,58.439,-72.201,171.982,28.570,155.287
C06060=1061.981,58.189,-72.183,171.981,28.567,155.286
C06061=1061.975,57.940,-72.166,171.979,28.565,155.286
C06062=1061.969,57.691,-72.150,171.978,28.562,155.286
C06063=1061.963,57.441,-72.132,171.977,28.559,155.285
C06064=1061.957,57.192,-72.116,171.975,28.557,155.285
C06065=1061.951,56.943,-72.099,171.973,28.554,155.285
C06066=1061.945,56.693,-72.081,171.972,28.551,155.284
C06067=1061.939,56.444,-72.064,171.970,28.549,155.284
C06068=1061.933,56.195,-72.048,171.970,28.547,155.283
C06069=1061.927,55.945,-72.030,171.968,28.544,155.283
C06070=1061.921,55.696,-72.014,171.966,28.541,155.283
C06071=1061.914,55.447,-71.997,171.965,28.538,155.282
C06072=1061.909,55.197,-71.980,171.963,28.536,155.282
C06073=1061.902,54.948,-71.963,171.961,28.533,155.282
C06074=1061.896,54.699,-71.947,171.961,28.531,155.281
C06075=1061.891,54.449,-71.929,171.959,28.528,155.281
C06076=1061.884,54.199,-71.912,171.958,28.526,155.280
C06077=1061.878,53.951,-71.895,171.956,28.523,155.280
C06078=1061.873,53.701,-71.878,171.954,28.520,155.280
C06079=1061.866,53.452,-71.862,171.953,28.517,155.279
C06080=1061.860,53.202,-71.845,171.952,28.515,155.279
C06081=1061.854,52.953,-71.827,171.950,28.513,155.279
C06082=1061.848,52.704,-71.811,171.949,28.510,155.278
C06083=1061.843,52.455,-71.795,171.947,28.507,155.278
C06084=1061.836,52.205,-71.777,171.946,28.505,155.278
C06085=1061.830,51.955,-71.761,171.945,28.502,155.277
C06086=1061.824,51.707,-71.744,171.943,28.500,155.277
C06087=1061.819,51.457,-71.727,171.942,28.497,155.276
C06088=1061.813,51.208,-71.711,171.940,28.494,155.276
C06089=1061.806,50.958,-71.693,171.939,28.492,155.276
C06090=1061.800,50.709,-71.677,171.937,28.489,155.275
C06091=1061.795,50.459,-71.660,171.936,28.486,155.275
C06092=1061.789,50.211,-71.643,171.935,28.484,155.274
C06093=1061.783,49.961,-71.627,171.933,28.481,155.274
C06094=1061.777,49.711,-71.610,171.931,28.479,155.274
C06095=1061.771,49.462,-71.593,171.930,28.476,155.273
C06096=1061.765,49.213,-71.576,171.928,28.473,155.273
C06097=1061.759,48.963,-71.560,171.928,28.470,155.273
C06098=1061.753,48.714,-71.543,171.926,28.468,155.272
C06099=1061.747,48.464,-71.526,171.924,28.465,155.272
C06100=1061.741,48.215,-71.510,171.923,28.463,155.271
C06101=1061.735,47.966,-71.493,171.921,28.460,155.271
C06102=1061.729,47.717,-71.476,171.921,28.457,155.271
C06103=1061.723,47.467,-71.460,171.919,28.455,155.270
C06104=1061.717,47.218,-71.443,171.917,28.452,155.270
C06105=1061.712,46.968,-71.427,171.916,28.450,155.270
C06106=1061.705,46.719,-71.409,171.914,28.447,155.269
C06107=1061.699,46.435,-71.391,171.913,28.444,155.269
C06108=1061.692,46.150,-71.372,171.911,28.441,155.268
C06109=1061.685,45.865,-71.353,171.909,28.438,155.268
C06110=1061.679,45.581,-71.334,171.908,28.435,155.267
C06111=1061.673,45.332,-71.318,171.906,28.432,155.267
C06112=1061.667,45.082,-71.301,171.905,28.429,155.267
C06113=1061.661,44.833,-71.284,171.903,28.427,155.266
C06114=1061.655,44.584,-71.268,171.902,28.425,155.266
C06115=1061.649,44.334,-71.251,171.901,28.422,155.266
C06116=1061.644,44.085,-71.235,171.899,28.419,155.265
C06117=1061.638,43.835,-71.218,171.898,28.416,155.265
C06118=1061.632,43.586,-71.202,171.896,28.413,155.264
C06119=1061.626,43.336,-71.186,171.895,28.411,155.264
C06120=1061.620,43.087,-71.170,171.894,28.409,155.264
C06121=1061.613,42.838,-71.152,171.892,28.406,155.263
C06122=1061.607,42.588,-71.136,171.890,28.404,155.263
C06123=1061.601,42.339,-71.120,171.889,28.401,155.263
C06124=1061.595,42.090,-71.103,171.887,28.398,155.262
C06125=1061.589,41.840,-71.087,171.887,28.396,155.262
C06126=1061.583,41.591,-71.071,171.885,28.393,155.262
C06127=1061.577,41.342,-71.055,171.883,28.391,155.261
C06128=1061.571,41.092,-71.038,171.882,28.388,155.261
C06129=1061.565,40.843,-71.022,171.880,28.385,155.260
C06130=1061.559,40.593,-71.005,171.879,28.383,155.260
C06131=1061.553,40.343,-70.989,171.878,28.380,155.260
C06132=1061.547,40.094,-70.973,171.876,28.378,155.259
C06133=1061.541,39.845,-70.957,171.875,28.375,155.259
C06134=1061.535,39.595,-70.940,171.873,28.372,155.259
C06135=1061.529,39.346,-70.924,171.871,28.370,155.258
C06136=1061.523,39.097,-70.908,171.870,28.367,155.258
C06137=1061.517,38.847,-70.892,171.869,28.365,155.257
C06138=1061.511,38.598,-70.875,171.868,28.362,155.257
C06139=1061.505,38.349,-70.859,171.866,28.360,155.257
C06140=1061.499,38.099,-70.843,171.864,28.357,155.256
C06141=1061.493,37.850,-70.827,171.863,28.354,155.256
C06142=1061.487,37.601,-70.810,171.861,28.352,155.256
C06143=1061.481,37.351,-70.794,171.861,28.349,155.255
C06144=1061.475,37.102,-70.778,171.859,28.347,155.255
C06145=1061.469,36.852,-70.763,171.857,28.344,155.255
C06146=1061.463,36.602,-70.746,171.856,28.342,155.254
C06147=1061.457,36.353,-70.730,171.854,28.339,155.254
C06148=1061.451,36.104,-70.714,171.853,28.336,155.254
C06149=1061.445,35.854,-70.698,171.852,28.335,155.253
C06150=1061.438,35.605,-70.682,171.850,28.332,155.253
C06151=1061.432,35.356,-70.666,171.849,28.329,155.253
C06152=1061.426,35.106,-70.650,171.847,28.327,155.252
C06153=1061.420,34.857,-70.634,171.845,28.324,155.252
C06154=1061.414,34.607,-70.618,171.844,28.321,155.251
C06155=1061.408,34.358,-70.602,171.843,28.319,155.251
C06156=1061.402,34.109,-70.586,171.842,28.316,155.251
C06157=1061.396,33.859,-70.569,171.840,28.314,155.250
C06158=1061.390,33.609,-70.554,171.838,28.311,155.250
C06159=1061.384,33.360,-70.538,171.837,28.308,155.250
C06160=1061.378,33.111,-70.522,171.835,28.306,155.249
C06161=1061.372,32.862,-70.506,171.834,28.304,155.249
C06162=1061.366,32.612,-70.490,171.833,28.301,155.249
C06163=1061.359,32.363,-70.475,171.831,28.299,155.248
C06164=1061.353,32.113,-70.458,171.830,28.296,155.248
C06165=1061.347,31.864,-70.442,171.828,28.294,155.248
C06166=1061.342,31.614,-70.426,171.826,28.291,155.247
C06167=1061.336,31.365,-70.410,171.826,28.289,155.247
C06168=1061.329,31.116,-70.395,171.824,28.286,155.247
C06169=1061.323,30.866,-70.378,171.823,28.283,155.246
C06170=1061.318,30.616,-70.363,171.821,28.281,155.246
C06171=1061.310,30.332,-70.345,171.819,28.278,155.246
C06172=1061.304,30.048,-70.327,171.818,28.275,155.245
C06173=1061.296,29.763,-70.308,171.816,28.272,155.245
C06174=1061.290,29.478,-70.290,171.815,28.269,155.244
C06175=1061.284,29.229,-70.274,171.813,28.267,155.244
C06176=1061.277,28.980,-70.259,171.811,28.264,155.244
C06177=1061.272,28.730,-70.243,171.810,28.261,155.243
C06178=1061.266,28.481,-70.227,171.808,28.259,155.243
C06179=1061.260,28.232,-70.212,171.807,28.256,155.243
C06180=1061.254,27.982,-70.196,171.806,28.254,155.242
C06181=1061.247,27.733,-70.180,171.804,28.252,155.242
C06182=1061.242,27.483,-70.165,171.803,28.249,155.242
C06183=1061.236,27.234,-70.148,171.801,28.246,155.241
C06184=1061.229,26.984,-70.134,171.800,28.244,155.241
C06185=1061.223,26.735,-70.117,171.798,28.241,155.240
C06186=1061.217,26.486,-70.102,171.797,28.239,155.240
C06187=1061.211,26.236,-70.086,171.796,28.237,155.240
C06188=1061.205,25.987,-70.070,171.794,28.234,155.239
C06189=1061.199,25.737,-70.055,171.792,28.232,155.239
C06190=1061.193,25.488,-70.039,171.791,28.229,155.239
C06191=1061.186,25.238,-70.024,171.789,28.227,155.238
C06192=1061.181,24.989,-70.007,171.788,28.224,155.238
C06193=1061.175,24.740,-69.993,171.787,28.222,155.238
C06194=1061.169,24.490,-69.977,171.785,28.219,155.237
C06195=1061.162,24.241,-69.962,171.784,28.217,155.237
C06196=1061.156,23.991,-69.945,171.782,28.214,155.237
C06197=1061.150,23.742,-69.930,171.781,28.212,155.236
C06198=1061.144,23.492,-69.914,171.779,28.209,155.236
C06199=1061.138,23.243,-69.899,171.778,28.207,155.236
C06200=1061.132,22.993,-69.883,171.777,28.204,155.235
C06201=1061.126,22.744,-69.868,171.775,28.202,155.235
C06202=1061.120,22.494,-69.853,171.773,28.199,155.235
C06203=1061.114,22.245,-69.837,171.772,28.197,155.234
C06204=1061.108,21.995,-69.822,171.770,28.194,155.234
C06205=1061.101,21.746,-69.806,171.769,28.192,155.234
C06206=1061.096,21.496,-69.790,171.768,28.189,155.233
C06207=1061.089,21.247,-69.775,171.766,28.187,155.233
C06208=1061.084,20.998,-69.760,171.765,28.184,155.233
C06209=1061.078,20.748,-69.745,171.763,28.181,155.232
C06210=1061.072,20.499,-69.728,171.762,28.179,155.232
C06211=1061.065,20.249,-69.713,171.760,28.176,155.232
C06212=1061.060,19.999,-69.698,171.759,28.174,155.231
C06213=1061.053,19.750,-69.682,171.758,28.172,155.231
C06214=1061.048,19.501,-69.667,171.756,28.169,155.231
C06215=1061.041,19.251,-69.652,171.754,28.167,155.230
C06216=1061.035,19.002,-69.636,171.753,28.164,155.230
C06217=1061.029,18.752,-69.621,171.751,28.162,155.230
C06218=1061.023,18.503,-69.606,171.750,28.159,155.229
C06219=1061.016,18.254,-69.590,171.749,28.157,155.229
C06220=1061.011,18.004,-69.575,171.747,28.154,155.229
C06221=1061.005,17.755,-69.560,171.746,28.152,155.228
C06222=1060.998,17.505,-69.545,171.744,28.149,155.228
C06223=1060.992,17.256,-69.529,171.743,28.147,155.228
C06224=1060.986,17.006,-69.514,171.741,28.145,155.227
C06225=1060.981,16.757,-69.499,171.739,28.142,155.227
C06226=1060.974,16.508,-69.483,171.739,28.140,155.227
C06227=1060.968,16.258,-69.468,171.737,28.137,155.226
C06228=1060.962,16.008,-69.453,171.735,28.135,155.226
C06229=1060.956,15.759,-69.438,171.734,28.132,155.226
C06230=1060.950,15.510,-69.423,171.732,28.130,155.225
C06231=1060.944,15.260,-69.407,171.731,28.127,155.225
C06232=1060.938,15.011,-69.392,171.729,28.125,155.225
C06233=1060.932,14.762,-69.377,171.728,28.122,155.224
C06234=1060.926,14.512,-69.362,171.727,28.120,155.224
C06235=1060.919,14.229,-69.345,171.725,28.117,155.224
C06236=1060.912,13.946,-69.327,171.723,28.114,155.223
C06237=1060.905,13.662,-69.311,171.721,28.112,155.223
C06238=1060.898,13.379,-69.294,171.720,28.109,155.223
C06239=1060.891,13.130,-69.279,171.718,28.106,155.222
C06240=1060.886,12.880,-69.263,171.716,28.104,155.222
C06241=1060.879,12.630,-69.248,171.716,28.102,155.222
C06242=1060.874,12.381,-69.234,171.714,28.100,155.221
C06243=1060.867,12.132,-69.218,171.712,28.097,155.221
C06244=1060.860,11.882,-69.203,171.711,28.095,155.221
C06245=1060.854,11.633,-69.188,171.709,28.093,155.220
C06246=1060.848,11.383,-69.173,171.708,28.090,155.220
C06247=1060.842,11.134,-69.159,171.706,28.087,155.220
C06248=1060.836,10.884,-69.143,171.704,28.085,155.220
C06249=1060.830,10.634,-69.128,171.704,28.083,155.219
C06250=1060.824,10.385,-69.114,171.702,28.080,155.219
C06251=1060.818,10.136,-69.099,171.700,28.078,155.219
C06252=1060.811,9.886,-69.084,171.699,28.075,155.218
C06253=1060.805,9.637,-69.069,171.697,28.073,155.218
C06254=1060.799,9.388,-69.054,171.696,28.071,155.218
C06255=1060.793,9.138,-69.039,171.694,28.068,155.217
C06256=1060.786,8.888,-69.024,171.692,28.066,155.217
C06257=1060.780,8.639,-69.009,171.692,28.064,155.217
C06258=1060.774,8.390,-68.995,171.690,28.061,155.216
C06259=1060.769,8.140,-68.979,171.689,28.059,155.216
C06260=1060.762,7.890,-68.964,171.687,28.057,155.216
C06261=1060.756,7.641,-68.950,171.685,28.054,155.215
C06262=1060.750,7.391,-68.935,171.684,28.051,155.215
C06263=1060.744,7.142,-68.920,171.682,28.049,155.215
C06264=1060.738,6.893,-68.905,171.680,28.047,155.215
C06265=1060.732,6.643,-68.890,171.680,28.044,155.214
C06266=1060.725,6.393,-68.875,171.678,28.042,155.214
C06267=1060.720,6.144,-68.861,171.677,28.040,155.214
C06268=1060.713,5.894,-68.846,171.675,28.037,155.213
C06269=1060.707,5.645,-68.832,171.673,28.035,155.213
C06270=1060.701,5.396,-68.817,171.672,28.033,155.213
C06271=1060.695,5.146,-68.802,171.670,28.030,155.212
C06272=1060.689,4.897,-68.787,171.669,28.028,155.212
C06273=1060.683,4.647,-68.772,171.668,28.026,155.212
C06274=1060.677,4.397,-68.757,171.666,28.023,155.211
C06275=1060.671,4.148,-68.743,171.665,28.020,155.211
C06276=1060.665,3.898,-68.728,171.663,28.018,155.211
C06277=1060.659,3.648,-68.713,171.661,28.016,155.210
C06278=1060.653,3.400,-68.699,171.660,28.013,155.210
C06279=1060.646,3.150,-68.684,171.658,28.011,155.210
C06280=1060.641,2.901,-68.669,171.657,28.009,155.210
C06281=1060.635,2.651,-68.655,171.655,28.006,155.209
C06282=1060.629,2.402,-68.640,171.654,28.004,155.209
C06283=1060.622,2.152,-68.625,171.653,28.002,155.209
C06284=1060.616,1.902,-68.610,171.651,27.999,155.208
C06285=1060.610,1.653,-68.596,171.649,27.997,155.208
C06286=1060.604,1.403,-68.582,171.648,27.994,155.208
C06287=1060.598,1.154,-68.567,171.646,27.992,155.207
C06288=1060.592,0.905,-68.552,171.645,27.989,155.207
C06289=1060.586,0.656,-68.537,171.643,27.987,155.207
C06290=1060.580,0.405,-68.523,171.641,27.985,155.206
C06291=1060.574,0.156,-68.508,171.641,27.982,155.206
C06292=1060.568,-0.093,-68.494,171.639,27.980,155.206
C06293=1060.562,-0.344,-68.479,171.638,27.978,155.205
C06294=1060.556,-0.593,-68.465,171.636,27.975,155.205
C06295=1060.550,-0.842,-68.450,171.634,27.973,155.205
C06296=1060.544,-1.091,-68.435,171.633,27.970,155.205
C06297=1060.538,-1.341,-68.421,171.631,27.968,155.204
C06298=1060.532,-1.590,-68.407,171.630,27.965,155.204
C06299=1060.525,-1.871,-68.391,171.628,27.963,155.204
C06300=1060.518,-2.154,-68.374,171.626,27.960,155.203
C06301=1060.512,-2.434,-68.357,171.625,27.957,155.203
C06302=1060.505,-2.716,-68.341,171.623,27.955,155.203
C06303=1060.499,-2.964,-68.327,171.622,27.952,155.202
C06304=1060.493,-3.215,-68.313,171.620,27.950,155.202
C06305=1060.487,-3.464,-68.298,171.618,27.948,155.202
C06306=1060.481,-3.714,-68.284,171.617,27.946,155.201
C06307=1060.474,-3.963,-68.269,171.615,27.943,155.201
C06308=1060.468,-4.212,-68.255,171.614,27.940,155.201
C06309=1060.462,-4.463,-68.241,171.613,27.938,155.200
C06310=1060.456,-4.711,-68.227,171.611,27.936,155.200
C06311=1060.450,-4.961,-68.212,171.610,27.934,155.200
C06312=1060.444,-5.210,-68.198,171.608,27.932,155.200
C06313=1060.438,-5.461,-68.184,171.606,27.929,155.199
C06314=1060.431,-5.709,-68.170,171.605,27.927,155.199
C06315=1060.425,-5.960,-68.155,171.603,27.925,155.199
C06316=1060.419,-6.209,-68.141,171.601,27.923,155.199
C06317=1060.413,-6.459,-68.127,171.600,27.920,155.198
C06318=1060.407,-6.708,-68.113,171.598,27.918,155.198
C06319=1060.401,-6.958,-68.098,171.597,27.915,155.198
C06320=1060.394,-7.206,-68.084,171.596,27.913,155.197
C06321=1060.388,-7.457,-68.070,171.594,27.911,155.197
C06322=1060.382,-7.706,-68.056,171.593,27.909,155.197
C06323=1060.376,-7.956,-68.041,171.591,27.907,155.196
C06324=1060.370,-8.205,-68.027,171.589,27.904,155.196
C06325=1060.364,-8.455,-68.013,171.588,27.902,155.196
C06326=1060.358,-8.704,-67.998,171.586,27.900,155.196
C06327=1060.351,-8.954,-67.985,171.585,27.898,155.195
C06328=1060.346,-9.203,-67.971,171.583,27.895,155.195
C06329=1060.339,-9.453,-67.956,171.581,27.892,155.195
C06330=1060.333,-9.702,-67.943,171.580,27.890,155.194
C06331=1060.327,-9.951,-67.928,171.578,27.888,155.194
C06332=1060.321,-10.202,-67.914,171.577,27.886,155.194
C06333=1060.315,-10.451,-67.901,171.576,27.884,155.194
C06334=1060.309,-10.700,-67.886,171.574,27.881,155.193
C06335=1060.303,-10.950,-67.872,171.573,27.879,155.193
C06336=1060.297,-11.199,-67.859,171.571,27.877,155.193
C06337=1060.291,-11.449,-67.844,171.569,27.875,155.193
C06338=1060.284,-11.698,-67.830,171.568,27.872,155.192
C06339=1060.278,-11.948,-67.816,171.566,27.870,155.192
C06340=1060.272,-12.197,-67.802,171.564,27.868,155.192
C06341=1060.266,-12.447,-67.788,171.563,27.866,155.192
C06342=1060.260,-12.697,-67.774,171.561,27.863,155.191
C06343=1060.254,-12.946,-67.759,171.560,27.861,155.191
C06344=1060.248,-13.196,-67.746,171.559,27.859,155.191
C06345=1060.242,-13.445,-67.732,171.557,27.856,155.190
C06346=1060.236,-13.694,-67.717,171.556,27.854,155.190
C06347=1060.230,-13.944,-67.704,171.554,27.852,155.190
C06348=1060.224,-14.194,-67.690,171.552,27.850,155.189
C06349=1060.218,-14.443,-67.677,171.551,27.847,155.189
C06350=1060.211,-14.693,-67.662,171.549,27.845,155.189
C06351=1060.206,-14.942,-67.648,171.548,27.843,155.189
C06352=1060.200,-15.192,-67.635,171.546,27.841,155.188
C06353=1060.194,-15.442,-67.620,171.544,27.838,155.188
C06354=1060.187,-15.691,-67.607,171.543,27.836,155.188
C06355=1060.180,-15.941,-67.593,171.541,27.834,155.188
C06356=1060.175,-16.190,-67.579,171.539,27.832,155.187
C06357=1060.169,-16.439,-67.566,171.538,27.829,155.187
C06358=1060.163,-16.690,-67.551,171.536,27.827,155.187
C06359=1060.156,-16.939,-67.538,171.535,27.826,155.187
C06360=1060.151,-17.188,-67.524,171.534,27.823,155.186
C06361=1060.144,-17.438,-67.510,171.532,27.821,155.186
C06362=1060.138,-17.687,-67.497,171.531,27.819,155.186
C06363=1060.131,-17.968,-67.481,171.529,27.817,155.186
C06364=1060.124,-18.247,-67.466,171.527,27.813,155.185
C06365=1060.116,-18.526,-67.450,171.525,27.811,155.185
C06366=1060.111,-18.806,-67.435,171.523,27.809,155.185
C06367=1060.104,-19.056,-67.422,171.522,27.807,155.184
C06368=1060.097,-19.305,-67.408,171.520,27.804,155.184
C06369=1060.092,-19.554,-67.394,171.518,27.802,155.184
C06370=1060.085,-19.804,-67.380,171.517,27.800,155.184
C06371=1060.080,-20.054,-67.366,171.515,27.798,155.183
C06372=1060.073,-20.303,-67.353,171.513,27.796,155.183
C06373=1060.067,-20.553,-67.339,171.512,27.794,155.183
C06374=1060.061,-20.803,-67.325,171.510,27.791,155.183
C06375=1060.055,-21.052,-67.312,171.510,27.789,155.182
C06376=1060.049,-21.302,-67.298,171.508,27.787,155.182
C06377=1060.043,-21.551,-67.285,171.506,27.785,155.182
C06378=1060.036,-21.801,-67.271,171.505,27.783,155.182
C06379=1060.031,-22.050,-67.258,171.503,27.780,155.181
C06380=1060.024,-22.300,-67.244,171.501,27.778,155.181
C06381=1060.018,-22.550,-67.231,171.500,27.777,155.181
C06382=1060.012,-22.799,-67.217,171.498,27.774,155.181
C06383=1060.006,-23.048,-67.204,171.496,27.772,155.180
C06384=1060.000,-23.298,-67.190,171.495,27.770,155.180
C06385=1059.994,-23.548,-67.176,171.493,27.767,155.180
C06386=1059.988,-23.797,-67.163,171.492,27.765,155.180
C06387=1059.982,-24.046,-67.149,171.490,27.763,155.179
C06388=1059.976,-24.296,-67.136,171.488,27.761,155.179
C06389=1059.969,-24.546,-67.122,171.487,27.759,155.179
C06390=1059.963,-24.795,-67.109,171.485,27.757,155.179
C06391=1059.958,-25.045,-67.095,171.483,27.754,155.178
C06392=1059.952,-25.295,-67.082,171.482,27.752,155.178
C06393=1059.945,-25.544,-67.069,171.480,27.750,155.178
C06394=1059.939,-25.794,-67.055,171.478,27.748,155.178
C06395=1059.933,-26.044,-67.042,171.478,27.746,155.177
C06396=1059.927,-26.293,-67.028,171.476,27.744,155.177
C06397=1059.921,-26.542,-67.014,171.475,27.742,155.177
C06398=1059.915,-26.792,-67.001,171.473,27.739,155.177
C06399=1059.908,-27.042,-66.988,171.471,27.737,155.176
C06400=1059.902,-27.291,-66.975,171.470,27.736,155.176
C06401=1059.896,-27.541,-66.962,171.468,27.733,155.176
C06402=1059.891,-27.790,-66.948,171.466,27.731,155.176
C06403=1059.885,-28.040,-66.935,171.465,27.729,155.175
C06404=1059.878,-28.290,-66.921,171.463,27.727,155.175
C06405=1059.872,-28.539,-66.908,171.461,27.725,155.175
C06406=1059.866,-28.789,-66.895,171.460,27.723,155.175
C06407=1059.859,-29.038,-66.882,171.458,27.721,155.174
C06408=1059.853,-29.287,-66.869,171.457,27.719,155.174
C06409=1059.846,-29.537,-66.855,171.455,27.717,155.174
C06410=1059.840,-29.787,-66.842,171.453,27.715,155.174
C06411=1059.834,-30.036,-66.829,171.452,27.712,155.174
C06412=1059.829,-30.286,-66.815,171.450,27.711,155.173
C06413=1059.823,-30.536,-66.803,171.448,27.708,155.173
C06414=1059.816,-30.786,-66.789,171.447,27.706,155.173
C06415=1059.810,-31.035,-66.776,171.445,27.705,155.173
C06416=1059.804,-31.284,-66.762,171.443,27.702,155.172
C06417=1059.798,-31.534,-66.750,171.442,27.700,155.172
C06418=1059.792,-31.783,-66.737,171.440,27.698,155.172
C06419=1059.785,-32.033,-66.723,171.438,27.696,155.172
C06420=1059.779,-32.283,-66.711,171.437,27.694,155.172
C06421=1059.773,-32.533,-66.697,171.435,27.692,155.171
C06422=1059.766,-32.782,-66.684,171.433,27.690,155.171
C06423=1059.760,-33.032,-66.671,171.432,27.688,155.171
C06424=1059.754,-33.281,-66.658,171.430,27.686,155.171
C06425=1059.749,-33.531,-66.644,171.428,27.684,155.170
C06426=1059.743,-33.780,-66.632,171.427,27.681,155.170
C06427=1059.735,-34.059,-66.617,171.425,27.680,155.170
C06428=1059.729,-34.338,-66.603,171.424,27.677,155.170
C06429=1059.722,-34.617,-66.588,171.422,27.675,155.169
C06430=1059.715,-34.896,-66.574,171.420,27.673,155.169
C06431=1059.709,-35.145,-66.561,171.419,27.671,155.169
C06432=1059.702,-35.395,-66.547,171.417,27.668,155.169
C06433=1059.697,-35.644,-66.535,171.415,27.667,155.169
C06434=1059.690,-35.894,-66.521,171.414,27.664,155.168
C06435=1059.685,-36.144,-66.508,171.412,27.663,155.168
C06436=1059.679,-36.393,-66.495,171.410,27.660,155.168
C06437=1059.673,-36.643,-66.482,171.409,27.658,155.168
C06438=1059.667,-36.892,-66.469,171.407,27.656,155.167
C06439=1059.661,-37.142,-66.457,171.406,27.654,155.167
C06440=1059.655,-37.391,-66.443,171.404,27.653,155.167
C06441=1059.649,-37.641,-66.430,171.402,27.650,155.167
C06442=1059.643,-37.891,-66.418,171.401,27.648,155.166
C06443=1059.637,-38.140,-66.405,171.399,27.646,155.166
C06444=1059.630,-38.390,-66.392,171.397,27.644,155.166
C06445=1059.625,-38.640,-66.379,171.396,27.642,155.166
C06446=1059.618,-38.890,-66.366,171.394,27.640,155.166
C06447=1059.611,-39.139,-66.354,171.392,27.638,155.166
C06448=1059.605,-39.388,-66.340,171.391,27.636,155.165
C06449=1059.599,-39.638,-66.328,171.389,27.634,155.165
C06450=1059.593,-39.888,-66.315,171.387,27.633,155.165
C06451=1059.587,-40.137,-66.302,171.386,27.630,155.165
C06452=1059.580,-40.387,-66.290,171.384,27.629,155.165
C06453=1059.574,-40.636,-66.277,171.382,27.627,155.164
C06454=1059.568,-40.886,-66.264,171.381,27.625,155.164
C06455=1059.562,-41.135,-66.251,171.379,27.623,155.164
C06456=1059.556,-41.385,-66.238,171.377,27.621,155.164
C06457=1059.549,-41.635,-66.226,171.376,27.619,155.164
C06458=1059.543,-41.884,-66.213,171.374,27.617,155.163
C06459=1059.537,-42.134,-66.201,171.372,27.615,155.163
C06460=1059.531,-42.384,-66.188,171.371,27.613,155.163
C06461=1059.525,-42.633,-66.175,171.369,27.611,155.163
C06462=1059.518,-42.883,-66.163,171.367,27.609,155.162
C06463=1059.513,-43.133,-66.150,171.366,27.607,155.162
C06464=1059.506,-43.382,-66.137,171.364,27.606,155.162
C06465=1059.500,-43.632,-66.124,171.362,27.603,155.162
C06466=1059.495,-43.882,-66.112,171.361,27.602,155.162
C06467=1059.488,-44.131,-66.099,171.359,27.599,155.162
C06468=1059.482,-44.381,-66.087,171.357,27.598,155.161
C06469=1059.476,-44.630,-66.074,171.356,27.596,155.161
C06470=1059.470,-44.880,-66.061,171.354,27.594,155.161
C06471=1059.463,-45.129,-66.049,171.352,27.592,155.161
C06472=1059.457,-45.379,-66.036,171.351,27.590,155.161
C06473=1059.452,-45.628,-66.024,171.349,27.588,155.160
C06474=1059.445,-45.878,-66.011,171.347,27.586,155.160
C06475=1059.439,-46.127,-65.999,171.346,27.584,155.160
C06476=1059.433,-46.377,-65.986,171.344,27.582,155.160
C06477=1059.427,-46.627,-65.974,171.342,27.581,155.160
C06478=1059.421,-46.877,-65.961,171.341,27.579,155.159
C06479=1059.414,-47.126,-65.949,171.339,27.577,155.159
C06480=1059.408,-47.376,-65.936,171.337,27.575,155.159
C06481=1059.402,-47.625,-65.923,171.336,27.573,155.159
C06482=1059.396,-47.875,-65.911,171.334,27.571,155.159
C06483=1059.390,-48.125,-65.899,171.332,27.569,155.159
C06484=1059.384,-48.373,-65.886,171.331,27.567,155.158
C06485=1059.378,-48.623,-65.873,171.329,27.566,155.158
C06486=1059.372,-48.873,-65.861,171.327,27.564,155.158
C06487=1059.366,-49.123,-65.849,171.326,27.562,155.158
C06488=1059.360,-49.373,-65.836,171.324,27.560,155.158
C06489=1059.354,-49.623,-65.824,171.322,27.558,155.157
C06490=1059.347,-49.872,-65.812,171.321,27.556,155.157
C06491=1059.341,-50.152,-65.797,171.318,27.554,155.157
C06492=1059.334,-50.431,-65.784,171.316,27.552,155.157
C06493=1059.326,-50.710,-65.770,171.315,27.550,155.157
C06494=1059.319,-50.989,-65.757,171.313,27.548,155.157
C06495=1059.314,-51.239,-65.745,171.311,27.546,155.156
C06496=1059.307,-51.488,-65.733,171.310,27.544,155.156
C06497=1059.302,-51.738,-65.720,171.308,27.543,155.156
C06498=1059.295,-51.988,-65.708,171.306,27.541,155.156
C06499=1059.288,-52.237,-65.696,171.304,27.539,155.156
C06500=1059.282,-52.486,-65.683,171.302,27.537,155.156
C06501=1059.275,-52.736,-65.671,171.300,27.536,155.155
C06502=1059.270,-52.986,-65.658,171.299,27.534,155.155
C06503=1059.263,-53.235,-65.646,171.297,27.532,155.155
C06504=1059.257,-53.486,-65.635,171.295,27.531,155.155
C06505=1059.251,-53.735,-65.623,171.293,27.529,155.155
C06506=1059.245,-53.984,-65.611,171.292,27.527,155.155
C06507=1059.239,-54.234,-65.598,171.290,27.525,155.154
C06508=1059.232,-54.484,-65.586,171.288,27.523,155.154
C06509=1059.226,-54.734,-65.574,171.287,27.522,155.154
C06510=1059.219,-54.983,-65.562,171.285,27.520,155.154
C06511=1059.213,-55.233,-65.550,171.283,27.518,155.154
C06512=1059.208,-55.482,-65.538,171.282,27.516,155.154
C06513=1059.201,-55.732,-65.526,171.280,27.515,155.154
C06514=1059.194,-55.981,-65.514,171.278,27.513,155.153
C06515=1059.188,-56.231,-65.501,171.277,27.511,155.153
C06516=1059.182,-56.481,-65.489,171.275,27.510,155.153
C06517=1059.176,-56.731,-65.477,171.273,27.508,155.153
C06518=1059.170,-56.980,-65.466,171.272,27.506,155.153
C06519=1059.163,-57.230,-65.454,171.270,27.505,155.153
C06520=1059.157,-57.479,-65.441,171.268,27.503,155.153
C06521=1059.151,-57.729,-65.429,171.266,27.501,155.152
C06522=1059.144,-57.979,-65.418,171.265,27.500,155.152
C06523=1059.139,-58.228,-65.405,171.263,27.498,155.152
C06524=1059.132,-58.477,-65.393,171.261,27.496,155.152
C06525=1059.126,-58.728,-65.382,171.260,27.494,155.152
C06526=1059.120,-58.977,-65.370,171.258,27.493,155.152
C06527=1059.114,-59.226,-65.358,171.255,27.491,155.152
C06528=1059.108,-59.476,-65.345,171.254,27.489,155.151
C06529=1059.101,-59.726,-65.333,171.252,27.487,155.151
C06530=1059.095,-59.976,-65.322,171.250,27.486,155.151
C06531=1059.090,-60.225,-65.310,171.248,27.484,155.151
C06532=1059.083,-60.475,-65.298,171.247,27.482,155.151
C06533=1059.076,-60.724,-65.286,171.245,27.481,155.151
C06534=1059.071,-60.975,-65.274,171.243,27.479,155.151
C06535=1059.065,-61.224,-65.263,171.242,27.477,155.150
C06536=1059.058,-61.473,-65.251,171.240,27.476,155.150
C06537=1059.052,-61.723,-65.238,171.238,27.474,155.150
C06538=1059.046,-61.973,-65.227,171.237,27.472,155.150
C06539=1059.040,-62.222,-65.215,171.235,27.471,155.150
C06540=1059.033,-62.472,-65.203,171.233,27.469,155.150
C06541=1059.028,-62.722,-65.192,171.231,27.468,155.150
C06542=1059.022,-62.971,-65.180,171.230,27.466,155.150
C06543=1059.015,-63.221,-65.168,171.228,27.464,155.149
C06544=1059.009,-63.471,-65.155,171.226,27.463,155.149
C06545=1059.003,-63.720,-65.145,171.225,27.461,155.149
C06546=1058.997,-63.970,-65.133,171.223,27.459,155.149
C06547=1058.991,-64.220,-65.120,171.221,27.458,155.149
C06548=1058.985,-64.469,-65.109,171.220,27.456,155.149
C06549=1058.978,-64.719,-65.097,171.218,27.454,155.149
C06550=1058.972,-64.969,-65.086,171.215,27.452,155.148
C06551=1058.967,-65.218,-65.074,171.214,27.451,155.148
C06552=1058.960,-65.468,-65.062,171.212,27.449,155.148
C06553=1058.954,-65.718,-65.051,171.210,27.448,155.148
C06554=1058.948,-65.967,-65.038,171.208,27.446,155.148
C06555=1058.941,-66.248,-65.026,171.207,27.444,155.148
C06556=1058.934,-66.528,-65.013,171.205,27.443,155.148
C06557=1058.928,-66.809,-64.999,171.202,27.441,155.148
C06558=1058.920,-67.089,-64.986,171.201,27.438,155.147
C06559=1058.915,-67.339,-64.975,171.199,27.437,155.147
C06560=1058.908,-67.588,-64.963,171.197,27.436,155.147
C06561=1058.903,-67.838,-64.951,171.196,27.434,155.147
C06562=1058.896,-68.088,-64.939,171.194,27.432,155.147
C06563=1058.890,-68.338,-64.928,171.192,27.431,155.147
C06564=1058.884,-68.587,-64.917,171.190,27.429,155.147
C06565=1058.878,-68.837,-64.905,171.189,27.428,155.147
C06566=1058.872,-69.086,-64.893,171.187,27.426,155.146
C06567=1058.866,-69.336,-64.882,171.185,27.424,155.146
C06568=1058.859,-69.586,-64.870,171.184,27.423,155.146
C06569=1058.854,-69.836,-64.858,171.182,27.421,155.146
C06570=1058.848,-70.085,-64.847,171.179,27.419,155.146
C06571=1058.842,-70.335,-64.836,171.177,27.418,155.146
C06572=1058.835,-70.584,-64.824,171.176,27.416,155.146
C06573=1058.830,-70.834,-64.812,171.174,27.415,155.146
C06574=1058.824,-71.084,-64.800,171.172,27.413,155.145
C06575=1058.818,-71.333,-64.789,171.171,27.412,155.145
C06576=1058.812,-71.583,-64.778,171.169,27.410,155.145
C06577=1058.805,-71.832,-64.767,171.167,27.408,155.145
C06578=1058.800,-72.083,-64.755,171.166,27.407,155.145
C06579=1058.794,-72.332,-64.743,171.164,27.405,155.145
C06580=1058.787,-72.582,-64.732,171.162,27.404,155.145
C06581=1058.782,-72.831,-64.721,171.160,27.402,155.145
C06582=1058.776,-73.081,-64.708,171.159,27.400,155.145
C06583=1058.770,-73.331,-64.698,171.157,27.399,155.144
C06584=1058.763,-73.580,-64.686,171.155,27.398,155.144
C06585=1058.758,-73.830,-64.675,171.153,27.396,155.144
C06586=1058.751,-74.080,-64.663,171.152,27.394,155.144
C06587=1058.745,-74.329,-64.652,171.150,27.393,155.144
C06588=1058.739,-74.579,-64.641,171.147,27.391,155.144
C06589=1058.733,-74.829,-64.630,171.146,27.390,155.144
C06590=1058.727,-75.079,-64.619,171.144,27.388,155.144
C06591=1058.721,-75.328,-64.607,171.142,27.387,155.144
C06592=1058.715,-75.578,-64.596,171.140,27.386,155.144
C06593=1058.709,-75.827,-64.585,171.139,27.384,155.143
C06594=1058.702,-76.077,-64.573,171.137,27.383,155.143
C06595=1058.696,-76.327,-64.562,171.135,27.381,155.143
C06596=1058.690,-76.577,-64.551,171.133,27.380,155.143
C06597=1058.684,-76.826,-64.540,171.132,27.378,155.143
C06598=1058.678,-77.076,-64.528,171.130,27.377,155.143
C06599=1058.672,-77.325,-64.517,171.128,27.375,155.143
C06600=1058.666,-77.575,-64.506,171.127,27.374,155.143
C06601=1058.660,-77.825,-64.495,171.125,27.373,155.143
C06602=1058.653,-78.075,-64.484,171.123,27.371,155.143
C06603=1058.647,-78.324,-64.472,171.120,27.370,155.143
C06604=1058.641,-78.574,-64.461,171.119,27.368,155.143
C06605=1058.635,-78.824,-64.450,171.117,27.367,155.143
C06606=1058.628,-79.073,-64.439,171.115,27.365,155.142
C06607=1058.623,-79.323,-64.428,171.113,27.364,155.142
C06608=1058.616,-79.572,-64.416,171.112,27.362,155.142
C06609=1058.610,-79.822,-64.406,171.110,27.361,155.142
C06610=1058.604,-80.072,-64.394,171.108,27.360,155.142
C06611=1058.598,-80.322,-64.383,171.106,27.358,155.142
C06612=1058.592,-80.572,-64.372,171.105,27.357,155.142
C06613=1058.585,-80.821,-64.362,171.103,27.356,155.142
C06614=1058.580,-81.070,-64.351,171.101,27.354,155.142
C06615=1058.573,-81.321,-64.340,171.099,27.353,155.142
C06616=1058.567,-81.570,-64.330,171.097,27.351,155.142
C06617=1058.560,-81.819,-64.318,171.095,27.350,155.142
C06618=1058.554,-82.069,-64.307,171.093,27.349,155.142
C06619=1058.547,-82.352,-64.295,171.091,27.347,155.142
C06620=1058.540,-82.635,-64.282,171.090,27.346,155.141
C06621=1058.533,-82.918,-64.270,171.087,27.344,155.141
C06622=1058.526,-83.200,-64.257,171.085,27.343,155.141
C06623=1058.519,-83.450,-64.247,171.083,27.342,155.141
C06624=1058.514,-83.700,-64.236,171.082,27.340,155.141
C06625=1058.507,-83.950,-64.225,171.080,27.339,155.141
C06626=1058.501,-84.199,-64.214,171.078,27.338,155.141
C06627=1058.495,-84.449,-64.203,171.075,27.337,155.141
C06628=1058.489,-84.699,-64.192,171.074,27.335,155.141
C06629=1058.483,-84.948,-64.181,171.072,27.334,155.141
C06630=1058.476,-85.198,-64.171,171.070,27.333,155.141
C06631=1058.470,-85.448,-64.160,171.068,27.332,155.141
C06632=1058.464,-85.697,-64.149,171.067,27.330,155.141
C06633=1058.457,-85.947,-64.138,171.065,27.329,155.141
C06634=1058.452,-86.196,-64.127,171.063,27.328,155.141
C06635=1058.445,-86.447,-64.116,171.061,27.327,155.141
C06636=1058.439,-86.696,-64.106,171.060,27.325,155.141
C06637=1058.433,-86.945,-64.095,171.058,27.324,155.141
C06638=1058.427,-87.196,-64.084,171.056,27.323,155.141
C06639=1058.421,-87.445,-64.074,171.053,27.322,155.141
C06640=1058.415,-87.695,-64.063,171.052,27.320,155.140
C06641=1058.409,-87.945,-64.052,171.050,27.319,155.140
C06642=1058.402,-88.194,-64.042,171.048,27.318,155.140
C06643=1058.396,-88.444,-64.031,171.046,27.316,155.140
C06644=1058.390,-88.694,-64.020,171.045,27.315,155.140
C06645=1058.383,-88.943,-64.009,171.043,27.314,155.140
C06646=1058.378,-89.193,-63.999,171.041,27.313,155.140
C06647=1058.372,-89.443,-63.988,171.039,27.311,155.140
C06648=1058.365,-89.692,-63.978,171.037,27.310,155.140
C06649=1058.359,-89.942,-63.967,171.036,27.309,155.140
C06650=1058.353,-90.192,-63.956,171.034,27.308,155.140
C06651=1058.347,-90.441,-63.945,171.031,27.307,155.140
C06652=1058.341,-90.691,-63.935,171.029,27.305,155.140
C06653=1058.335,-90.941,-63.925,171.028,27.304,155.140
C06654=1058.328,-91.191,-63.914,171.026,27.303,155.140
C06655=1058.323,-91.440,-63.903,171.024,27.302,155.140
C06656=1058.316,-91.689,-63.892,171.022,27.301,155.140
C06657=1058.311,-91.940,-63.882,171.021,27.299,155.140
C06658=1058.304,-92.190,-63.871,171.019,27.298,155.140
C06659=1058.298,-92.439,-63.861,171.017,27.297,155.140
C06660=1058.292,-92.688,-63.850,171.015,27.296,155.140
C06661=1058.286,-92.938,-63.840,171.013,27.294,155.140
C06662=1058.280,-93.188,-63.829,171.012,27.293,155.140
C06663=1058.274,-93.438,-63.818,171.009,27.292,155.140
C06664=1058.267,-93.687,-63.808,171.007,27.291,155.140
C06665=1058.262,-93.937,-63.798,171.005,27.290,155.140
C06666=1058.255,-94.187,-63.787,171.004,27.289,155.140
C06667=1058.249,-94.437,-63.776,171.002,27.288,155.139
C06668=1058.244,-94.687,-63.766,171.000,27.286,155.139
C06669=1058.237,-94.936,-63.756,170.998,27.285,155.139
C06670=1058.232,-95.185,-63.745,170.996,27.284,155.139
C06671=1058.225,-95.436,-63.735,170.995,27.283,155.139
C06672=1058.219,-95.685,-63.724,170.993,27.282,155.139
C06673=1058.213,-95.935,-63.713,170.991,27.281,155.139
C06674=1058.207,-96.185,-63.704,170.989,27.280,155.139
C06675=1058.201,-96.434,-63.693,170.987,27.278,155.139
C06676=1058.195,-96.683,-63.682,170.985,27.277,155.139
C06677=1058.189,-96.934,-63.672,170.983,27.276,155.139
C06678=1058.182,-97.183,-63.662,170.981,27.275,155.139
C06679=1058.177,-97.433,-63.651,170.979,27.274,155.139
C06680=1058.171,-97.683,-63.641,170.978,27.273,155.139
C06681=1058.165,-97.932,-63.630,170.976,27.272,155.139
C06682=1058.158,-98.183,-63.620,170.974,27.271,155.139
C06683=1058.151,-98.467,-63.608,170.971,27.269,155.139
C06684=1058.145,-98.752,-63.597,170.970,27.268,155.139
C06685=1058.137,-99.037,-63.586,170.968,27.267,155.139
C06686=1058.130,-99.322,-63.574,170.965,27.266,155.139
C06687=1058.124,-99.572,-63.564,170.963,27.265,155.139
C06688=1058.118,-99.822,-63.553,170.961,27.263,155.139
C06689=1058.111,-100.072,-63.543,170.960,27.263,155.139
C06690=1058.105,-100.321,-63.533,170.958,27.262,155.139
C06691=1058.099,-100.571,-63.523,170.956,27.261,155.139
C06692=1058.093,-100.820,-63.512,170.954,27.260,155.139
C06693=1058.087,-101.070,-63.503,170.952,27.258,155.139
C06694=1058.081,-101.320,-63.492,170.950,27.258,155.139
C06695=1058.074,-101.570,-63.482,170.948,27.257,155.139
C06696=1058.068,-101.819,-63.472,170.946,27.255,155.139
C06697=1058.062,-102.069,-63.462,170.944,27.254,155.139
C06698=1058.056,-102.319,-63.451,170.942,27.254,155.139
C06699=1058.050,-102.568,-63.442,170.941,27.253,155.139
C06700=1058.044,-102.819,-63.432,170.939,27.252,155.139
C06701=1058.038,-103.068,-63.421,170.937,27.250,155.139
C06702=1058.032,-103.318,-63.412,170.935,27.250,155.139
C06703=1058.025,-103.568,-63.401,170.933,27.249,155.139
C06704=1058.019,-103.818,-63.391,170.931,27.248,155.139
C06705=1058.013,-104.067,-63.381,170.929,27.246,155.139
C06706=1058.007,-104.317,-63.371,170.927,27.246,155.139
C06707=1058.001,-104.567,-63.361,170.925,27.245,155.139
C06708=1057.995,-104.816,-63.351,170.923,27.244,155.139
C06709=1057.988,-105.066,-63.341,170.921,27.243,155.139
C06710=1057.983,-105.316,-63.331,170.920,27.242,155.139
C06711=1057.977,-105.565,-63.321,170.918,27.241,155.139
C06712=1057.970,-105.815,-63.311,170.916,27.240,155.139
C06713=1057.965,-106.065,-63.301,170.914,27.239,155.139
C06714=1057.958,-106.314,-63.291,170.912,27.238,155.139
C06715=1057.952,-106.564,-63.281,170.910,27.237,155.140
C06716=1057.945,-106.814,-63.271,170.908,27.236,155.140
C06717=1057.939,-107.064,-63.262,170.906,27.235,155.140
C06718=1057.934,-107.314,-63.251,170.904,27.235,155.140
C06719=1057.927,-107.563,-63.241,170.902,27.234,155.140
C06720=1057.921,-107.813,-63.232,170.900,27.233,155.140
C06721=1057.915,-108.062,-63.221,170.899,27.232,155.140
C06722=1057.909,-108.312,-63.212,170.897,27.231,155.140
C06723=1057.902,-108.562,-63.202,170.895,27.230,155.140
C06724=1057.897,-108.812,-63.192,170.893,27.230,155.140
C06725=1057.891,-109.062,-63.182,170.890,27.228,155.140
C06726=1057.884,-109.311,-63.172,170.889,27.227,155.140
C06727=1057.878,-109.561,-63.163,170.887,27.227,155.140
C06728=1057.872,-109.811,-63.153,170.885,27.226,155.140
C06729=1057.866,-110.060,-63.143,170.883,27.225,155.140
C06730=1057.860,-110.310,-63.134,170.881,27.224,155.140
C06731=1057.853,-110.559,-63.124,170.879,27.223,155.140
C06732=1057.848,-110.809,-63.113,170.877,27.223,155.140
C06733=1057.842,-111.059,-63.104,170.876,27.222,155.140
C06734=1057.835,-111.309,-63.094,170.874,27.221,155.140
C06735=1057.829,-111.559,-63.085,170.871,27.220,155.140
C06736=1057.823,-111.809,-63.075,170.869,27.219,155.140
C06737=1057.817,-112.058,-63.065,170.867,27.218,155.140
C06738=1057.810,-112.308,-63.055,170.865,27.218,155.140
C06739=1057.804,-112.557,-63.046,170.864,27.217,155.140
C06740=1057.798,-112.807,-63.036,170.862,27.216,155.140
C06741=1057.792,-113.057,-63.027,170.860,27.215,155.140
C06742=1057.786,-113.307,-63.017,170.858,27.215,155.141
C06743=1057.780,-113.557,-63.007,170.856,27.214,155.141
C06744=1057.774,-113.807,-62.997,170.854,27.213,155.141
C06745=1057.768,-114.057,-62.988,170.853,27.212,155.141
C06746=1057.762,-114.306,-62.978,170.850,27.211,155.141
C06747=1057.755,-114.589,-62.967,170.848,27.211,155.141
C06748=1057.747,-114.873,-62.956,170.846,27.210,155.141
C06749=1057.740,-115.156,-62.945,170.843,27.209,155.141
C06750=1057.733,-115.440,-62.934,170.841,27.208,155.141
C06751=1057.727,-115.690,-62.925,170.840,27.208,155.141
C06752=1057.721,-115.939,-62.915,170.838,27.206,155.141
C06753=1057.715,-116.189,-62.906,170.836,27.206,155.141
C06754=1057.709,-116.438,-62.896,170.833,27.205,155.141
C06755=1057.703,-116.688,-62.887,170.831,27.204,155.141
C06756=1057.697,-116.938,-62.877,170.829,27.204,155.141
C06757=1057.691,-117.188,-62.868,170.827,27.203,155.142
C06758=1057.684,-117.438,-62.858,170.826,27.203,155.142
C06759=1057.678,-117.687,-62.848,170.824,27.201,155.142
C06760=1057.672,-117.938,-62.840,170.822,27.201,155.142
C06761=1057.666,-118.187,-62.831,170.820,27.200,155.142
C06762=1057.659,-118.437,-62.821,170.818,27.200,155.142
C06763=1057.653,-118.687,-62.811,170.816,27.199,155.142
C06764=1057.648,-118.936,-62.802,170.814,27.198,155.142
C06765=1057.641,-119.186,-62.793,170.812,27.197,155.142
C06766=1057.635,-119.436,-62.783,170.810,27.197,155.142
C06767=1057.629,-119.685,-62.774,170.808,27.196,155.142
C06768=1057.623,-119.935,-62.764,170.806,27.195,155.142
C06769=1057.617,-120.185,-62.754,170.804,27.195,155.142
C06770=1057.611,-120.435,-62.745,170.802,27.194,155.142
C06771=1057.604,-120.685,-62.737,170.800,27.194,155.143
C06772=1057.598,-120.934,-62.727,170.799,27.193,155.143
C06773=1057.592,-121.184,-62.718,170.797,27.193,155.143
C06774=1057.586,-121.434,-62.708,170.794,27.192,155.143
C06775=1057.580,-121.683,-62.699,170.792,27.191,155.143
C06776=1057.574,-121.933,-62.689,170.790,27.190,155.143
C06777=1057.568,-122.184,-62.680,170.788,27.190,155.143
C06778=1057.561,-122.433,-62.671,170.786,27.189,155.143
C06779=1057.555,-122.682,-62.662,170.784,27.189,155.143
C06780=1057.549,-122.932,-62.653,170.783,27.188,155.143
C06781=1057.543,-123.182,-62.643,170.781,27.188,155.143
C06782=1057.537,-123.432,-62.634,170.779,27.187,155.143
C06783=1057.531,-123.682,-62.625,170.777,27.187,155.144
C06784=1057.525,-123.931,-62.615,170.774,27.186,155.144
C06785=1057.519,-124.180,-62.606,170.772,27.185,155.144
C06786=1057.512,-124.430,-62.597,170.770,27.184,155.144
C06787=1057.506,-124.681,-62.588,170.769,27.184,155.144
C06788=1057.500,-124.931,-62.578,170.767,27.183,155.144
C06789=1057.493,-125.180,-62.569,170.765,27.183,155.144
C06790=1057.488,-125.430,-62.561,170.763,27.182,155.144
C06791=1057.482,-125.680,-62.551,170.761,27.182,155.144
C06792=1057.476,-125.929,-62.542,170.759,27.182,155.144
C06793=1057.469,-126.179,-62.533,170.757,27.181,155.145
C06794=1057.463,-126.429,-62.524,170.754,27.180,155.145
C06795=1057.457,-126.678,-62.515,170.752,27.180,155.145
C06796=1057.451,-126.928,-62.506,170.751,27.179,155.145
C06797=1057.445,-127.178,-62.497,170.749,27.179,155.145
C06798=1057.438,-127.428,-62.487,170.747,27.178,155.145
C06799=1057.433,-127.677,-62.478,170.745,27.178,155.145
C06800=1057.427,-127.928,-62.469,170.743,27.177,155.145
C06801=1057.422,-128.177,-62.460,170.741,27.176,155.145
C06802=1057.419,-128.427,-62.449,170.740,27.175,155.145
C06803=1057.417,-128.678,-62.438,170.738,27.172,155.145
C06804=1057.416,-128.929,-62.426,170.736,27.169,155.145
C06805=1057.417,-129.179,-62.413,170.735,27.166,155.144
C06806=1057.418,-129.430,-62.400,170.735,27.162,155.143
C06807=1057.421,-129.681,-62.386,170.734,27.157,155.143
C06808=1057.426,-129.933,-62.371,170.733,27.153,155.142
C06809=1057.432,-130.183,-62.356,170.732,27.147,155.141
C06810=1057.438,-130.433,-62.339,170.733,27.141,155.140
C06811=1057.064,-130.456,-62.543,170.684,27.304,155.173
C06812=1057.057,-130.206,-62.558,170.685,27.310,155.174
C06813=1057.051,-129.955,-62.574,170.685,27.316,155.175
C06814=1057.047,-129.704,-62.588,170.686,27.321,155.176
C06815=1057.043,-129.452,-62.603,170.686,27.325,155.177
C06816=1057.042,-129.202,-62.616,170.688,27.329,155.177
C06817=1057.041,-128.952,-62.629,170.689,27.333,155.178
C06818=1057.041,-128.701,-62.641,170.690,27.336,155.178
C06819=1057.044,-128.451,-62.652,170.692,27.338,155.178
C06820=1057.047,-128.201,-62.663,170.694,27.340,155.178
C06821=1057.051,-127.950,-62.673,170.696,27.341,155.178
C06822=1057.057,-127.700,-62.682,170.697,27.341,155.178
C06823=1057.063,-127.451,-62.692,170.699,27.342,155.178
C06824=1057.069,-127.201,-62.700,170.701,27.342,155.178
C06825=1057.075,-126.951,-62.709,170.703,27.343,155.178
C06826=1057.081,-126.702,-62.719,170.705,27.343,155.178
C06827=1057.088,-126.452,-62.727,170.707,27.344,155.178
C06828=1057.094,-126.202,-62.736,170.709,27.344,155.178
C06829=1057.100,-125.953,-62.746,170.711,27.345,155.178
C06830=1057.106,-125.702,-62.755,170.713,27.345,155.178
C06831=1057.113,-125.453,-62.764,170.715,27.346,155.178
C06832=1057.119,-125.203,-62.773,170.717,27.347,155.177
C06833=1057.124,-124.953,-62.782,170.719,27.347,155.177
C06834=1057.131,-124.704,-62.791,170.721,27.348,155.177
C06835=1057.137,-124.454,-62.800,170.723,27.348,155.177
C06836=1057.143,-124.204,-62.810,170.725,27.349,155.177
C06837=1057.149,-123.954,-62.819,170.727,27.349,155.177
C06838=1057.155,-123.704,-62.828,170.729,27.350,155.177
C06839=1057.162,-123.455,-62.837,170.730,27.350,155.177
C06840=1057.168,-123.205,-62.847,170.733,27.351,155.177
C06841=1057.174,-122.956,-62.856,170.735,27.351,155.177
C06842=1057.180,-122.705,-62.865,170.737,27.352,155.176
C06843=1057.186,-122.455,-62.875,170.739,27.352,155.176
C06844=1057.192,-122.206,-62.884,170.741,27.353,155.176
C06845=1057.198,-121.956,-62.893,170.743,27.353,155.176
C06846=1057.205,-121.707,-62.902,170.745,27.354,155.176
C06847=1057.211,-121.457,-62.911,170.746,27.355,155.176
C06848=1057.217,-121.207,-62.921,170.748,27.355,155.176
C06849=1057.223,-120.957,-62.930,170.751,27.356,155.176
C06850=1057.229,-120.707,-62.940,170.753,27.357,155.176
C06851=1057.235,-120.458,-62.949,170.755,27.357,155.176
C06852=1057.241,-120.208,-62.959,170.757,27.358,155.176
C06853=1057.247,-119.958,-62.968,170.759,27.359,155.176
C06854=1057.254,-119.708,-62.976,170.761,27.359,155.176
C06855=1057.260,-119.459,-62.986,170.762,27.360,155.175
C06856=1057.266,-119.209,-62.996,170.764,27.360,155.175
C06857=1057.272,-118.959,-63.005,170.766,27.361,155.175
C06858=1057.278,-118.709,-63.015,170.768,27.361,155.175
C06859=1057.284,-118.460,-63.024,170.771,27.363,155.175
C06860=1057.290,-118.210,-63.033,170.773,27.363,155.175
C06861=1057.296,-117.960,-63.043,170.775,27.364,155.175
C06862=1057.302,-117.711,-63.053,170.776,27.364,155.175
C06863=1057.309,-117.461,-63.062,170.778,27.365,155.175
C06864=1057.315,-117.211,-63.072,170.780,27.366,155.175
C06865=1057.321,-116.961,-63.081,170.782,27.366,155.175
C06866=1057.327,-116.711,-63.091,170.784,27.367,155.175
C06867=1057.334,-116.462,-63.100,170.786,27.368,155.175
C06868=1057.340,-116.212,-63.109,170.789,27.369,155.174
C06869=1057.346,-115.962,-63.119,170.790,27.369,155.174
C06870=1057.352,-115.713,-63.129,170.792,27.370,155.174
C06871=1057.359,-115.463,-63.138,170.794,27.371,155.174
C06872=1057.365,-115.179,-63.149,170.796,27.371,155.174
C06873=1057.372,-114.896,-63.160,170.799,27.373,155.174
C06874=1057.379,-114.612,-63.171,170.801,27.373,155.174
C06875=1057.386,-114.328,-63.182,170.803,27.374,155.174
C06876=1057.392,-114.079,-63.192,170.805,27.375,155.174
C06877=1057.398,-113.829,-63.201,170.807,27.376,155.174
C06878=1057.404,-113.580,-63.210,170.809,27.376,155.174
C06879=1057.410,-113.330,-63.220,170.811,27.377,155.174
C06880=1057.416,-113.080,-63.229,170.813,27.378,155.174
C06881=1057.423,-112.830,-63.239,170.815,27.379,155.174
C06882=1057.429,-112.580,-63.249,170.816,27.379,155.174
C06883=1057.435,-112.331,-63.258,170.818,27.380,155.174
C06884=1057.441,-112.081,-63.268,170.820,27.381,155.174
C06885=1057.448,-111.832,-63.278,170.822,27.382,155.174
C06886=1057.453,-111.582,-63.288,170.825,27.383,155.173
C06887=1057.459,-111.332,-63.298,170.827,27.383,155.173
C06888=1057.465,-111.082,-63.307,170.828,27.384,155.173
C06889=1057.471,-110.832,-63.317,170.830,27.385,155.173
C06890=1057.478,-110.582,-63.326,170.832,27.386,155.173
C06891=1057.484,-110.333,-63.337,170.834,27.387,155.173
C06892=1057.490,-110.083,-63.346,170.836,27.388,155.173
C06893=1057.496,-109.834,-63.356,170.838,27.388,155.173
C06894=1057.503,-109.584,-63.365,170.839,27.389,155.173
C06895=1057.508,-109.334,-63.376,170.842,27.390,155.173
C06896=1057.515,-109.085,-63.386,170.844,27.391,155.173
C06897=1057.521,-108.835,-63.395,170.846,27.392,155.173
C06898=1057.527,-108.585,-63.405,170.848,27.393,155.173
C06899=1057.534,-108.334,-63.415,170.850,27.393,155.173
C06900=1057.540,-108.085,-63.425,170.851,27.394,155.173
C06901=1057.546,-107.835,-63.435,170.853,27.395,155.173
C06902=1057.552,-107.586,-63.444,170.855,27.396,155.173
C06903=1057.558,-107.336,-63.455,170.857,27.397,155.173
C06904=1057.564,-107.086,-63.465,170.859,27.398,155.173
C06905=1057.571,-106.837,-63.474,170.862,27.398,155.173
C06906=1057.577,-106.587,-63.484,170.863,27.400,155.173
C06907=1057.582,-106.337,-63.495,170.865,27.401,155.173
C06908=1057.589,-106.087,-63.504,170.867,27.401,155.173
C06909=1057.595,-105.838,-63.514,170.869,27.402,155.173
C06910=1057.601,-105.588,-63.524,170.871,27.403,155.173
C06911=1057.607,-105.338,-63.534,170.873,27.404,155.173
C06912=1057.613,-105.089,-63.544,170.874,27.405,155.173
C06913=1057.619,-104.839,-63.554,170.876,27.406,155.173
C06914=1057.626,-104.590,-63.564,170.878,27.407,155.173
C06915=1057.632,-104.339,-63.574,170.881,27.408,155.173
C06916=1057.638,-104.090,-63.585,170.883,27.409,155.173
C06917=1057.644,-103.840,-63.594,170.885,27.410,155.172
C06918=1057.650,-103.590,-63.604,170.886,27.411,155.172
C06919=1057.656,-103.341,-63.615,170.888,27.412,155.173
C06920=1057.662,-103.091,-63.624,170.890,27.413,155.173
C06921=1057.668,-102.841,-63.635,170.892,27.413,155.172
C06922=1057.674,-102.591,-63.645,170.894,27.414,155.172
C06923=1057.681,-102.342,-63.655,170.895,27.416,155.172
C06924=1057.687,-102.091,-63.665,170.897,27.417,155.173
C06925=1057.693,-101.842,-63.675,170.900,27.417,155.172
C06926=1057.699,-101.592,-63.685,170.902,27.419,155.172
C06927=1057.705,-101.342,-63.695,170.904,27.420,155.172
C06928=1057.711,-101.093,-63.706,170.905,27.421,155.172
C06929=1057.717,-100.843,-63.715,170.907,27.421,155.172
C06930=1057.723,-100.594,-63.726,170.909,27.422,155.172
C06931=1057.730,-100.343,-63.736,170.911,27.423,155.172
C06932=1057.736,-100.094,-63.746,170.913,27.425,155.172
C06933=1057.742,-99.844,-63.757,170.914,27.426,155.172
C06934=1057.748,-99.595,-63.767,170.916,27.426,155.172
C06935=1057.755,-99.345,-63.776,170.919,27.428,155.172
C06936=1057.762,-99.060,-63.789,170.921,27.429,155.172
C06937=1057.769,-98.775,-63.801,170.923,27.430,155.172
C06938=1057.776,-98.489,-63.812,170.925,27.431,155.172
C06939=1057.783,-98.205,-63.824,170.927,27.432,155.172
C06940=1057.788,-97.955,-63.834,170.929,27.433,155.172
C06941=1057.796,-97.705,-63.844,170.931,27.434,155.172
C06942=1057.801,-97.455,-63.855,170.933,27.435,155.172
C06943=1057.807,-97.206,-63.865,170.935,27.436,155.172
C06944=1057.813,-96.956,-63.876,170.937,27.437,155.172
C06945=1057.819,-96.706,-63.885,170.939,27.438,155.172
C06946=1057.825,-96.457,-63.896,170.941,27.440,155.172
C06947=1057.832,-96.207,-63.907,170.943,27.441,155.172
C06948=1057.838,-95.957,-63.917,170.944,27.442,155.172
C06949=1057.843,-95.707,-63.928,170.946,27.443,155.173
C06950=1057.850,-95.458,-63.938,170.948,27.445,155.173
C06951=1057.855,-95.208,-63.948,170.950,27.446,155.173
C06952=1057.862,-94.959,-63.959,170.951,27.447,155.173
C06953=1057.868,-94.709,-63.970,170.953,27.448,155.173
C06954=1057.874,-94.459,-63.979,170.956,27.449,155.173
C06955=1057.880,-94.209,-63.990,170.958,27.450,155.173
C06956=1057.886,-93.960,-64.001,170.960,27.451,155.173
C06957=1057.893,-93.709,-64.011,170.961,27.453,155.173
C06958=1057.898,-93.460,-64.022,170.963,27.454,155.173
C06959=1057.905,-93.211,-64.032,170.965,27.455,155.173
C06960=1057.910,-92.961,-64.043,170.967,27.456,155.173
C06961=1057.916,-92.711,-64.053,170.969,27.457,155.173
C06962=1057.923,-92.461,-64.064,170.970,27.458,155.173
C06963=1057.929,-92.212,-64.075,170.972,27.459,155.173
C06964=1057.934,-91.962,-64.086,170.974,27.460,155.173
C06965=1057.941,-91.712,-64.095,170.976,27.462,155.173
C06966=1057.947,-91.462,-64.106,170.978,27.463,155.173
C06967=1057.953,-91.213,-64.117,170.980,27.464,155.173
C06968=1057.959,-90.964,-64.128,170.982,27.466,155.173
C06969=1057.966,-90.713,-64.139,170.984,27.467,155.173
C06970=1057.972,-90.464,-64.148,170.985,27.468,155.173
C06971=1057.977,-90.214,-64.159,170.987,27.469,155.173
C06972=1057.983,-89.965,-64.170,170.989,27.470,155.173
C06973=1057.990,-89.715,-64.181,170.991,27.472,155.173
C06974=1057.996,-89.465,-64.192,170.993,27.473,155.173
C06975=1058.002,-89.216,-64.203,170.994,27.474,155.173
C06976=1058.009,-88.965,-64.213,170.996,27.475,155.173
C06977=1058.014,-88.716,-64.223,170.999,27.476,155.173
C06978=1058.020,-88.466,-64.234,171.001,27.477,155.173
C06979=1058.027,-88.216,-64.245,171.002,27.479,155.174
C06980=1058.033,-87.967,-64.256,171.004,27.480,155.174
C06981=1058.039,-87.718,-64.266,171.006,27.481,155.174
C06982=1058.046,-87.468,-64.277,171.008,27.482,155.174
C06983=1058.051,-87.218,-64.288,171.010,27.483,155.174
C06984=1058.058,-86.969,-64.298,171.011,27.485,155.174
C06985=1058.064,-86.718,-64.309,171.013,27.486,155.174
C06986=1058.070,-86.469,-64.320,171.015,27.487,155.174
C06987=1058.075,-86.219,-64.331,171.017,27.488,155.174
C06988=1058.082,-85.969,-64.341,171.018,27.490,155.174
C06989=1058.088,-85.720,-64.352,171.021,27.492,155.174
C06990=1058.095,-85.470,-64.364,171.023,27.493,155.174
C06991=1058.101,-85.220,-64.374,171.025,27.494,155.174
C06992=1058.107,-84.971,-64.385,171.026,27.495,155.174
C06993=1058.113,-84.721,-64.396,171.028,27.497,155.174
C06994=1058.120,-84.471,-64.406,171.030,27.498,155.174
C06995=1058.126,-84.221,-64.417,171.032,27.499,155.174
C06996=1058.132,-83.972,-64.428,171.034,27.500,155.174
C06997=1058.138,-83.723,-64.439,171.035,27.502,155.174
C06998=1058.144,-83.472,-64.450,171.037,27.503,155.174
C06999=1058.150,-83.223,-64.461,171.039,27.504,155.175
C07000=1058.158,-82.941,-64.473,171.041,27.506,155.175
C07001=1058.164,-82.657,-64.485,171.043,27.507,155.175
C07002=1058.172,-82.374,-64.498,171.046,27.509,155.175
C07003=1058.179,-82.091,-64.511,171.048,27.510,155.175
C07004=1058.185,-81.842,-64.521,171.050,27.511,155.175
C07005=1058.191,-81.592,-64.532,171.051,27.513,155.175
C07006=1058.198,-81.343,-64.544,171.053,27.514,155.175
C07007=1058.203,-81.093,-64.554,171.055,27.515,155.175
C07008=1058.210,-80.843,-64.565,171.056,27.517,155.175
C07009=1058.216,-80.594,-64.576,171.058,27.518,155.175
C07010=1058.222,-80.344,-64.587,171.060,27.519,155.175
C07011=1058.228,-80.094,-64.598,171.063,27.521,155.175
C07012=1058.235,-79.844,-64.609,171.065,27.522,155.175
C07013=1058.241,-79.595,-64.620,171.066,27.523,155.175
C07014=1058.248,-79.345,-64.632,171.068,27.525,155.175
C07015=1058.253,-79.096,-64.643,171.070,27.526,155.175
C07016=1058.260,-78.845,-64.654,171.072,27.527,155.176
C07017=1058.265,-78.596,-64.665,171.073,27.528,155.176
C07018=1058.272,-78.346,-64.676,171.075,27.530,155.176
C07019=1058.278,-78.096,-64.687,171.077,27.531,155.176
C07020=1058.284,-77.847,-64.699,171.079,27.533,155.176
C07021=1058.290,-77.597,-64.710,171.080,27.534,155.176
C07022=1058.296,-77.347,-64.721,171.082,27.536,155.176
C07023=1058.302,-77.098,-64.732,171.084,27.537,155.176
C07024=1058.308,-76.849,-64.743,171.085,27.539,155.176
C07025=1058.314,-76.599,-64.755,171.088,27.540,155.176
C07026=1058.320,-76.349,-64.765,171.090,27.542,155.176
C07027=1058.326,-76.099,-64.777,171.092,27.543,155.177
C07028=1058.333,-75.850,-64.788,171.093,27.544,155.177
C07029=1058.340,-75.600,-64.799,171.095,27.546,155.177
C07030=1058.346,-75.350,-64.810,171.097,27.547,155.177
C07031=1058.352,-75.101,-64.822,171.099,27.549,155.177
C07032=1058.358,-74.851,-64.833,171.100,27.550,155.177
C07033=1058.364,-74.601,-64.844,171.102,27.552,155.177
C07034=1058.370,-74.351,-64.855,171.104,27.553,155.177
C07035=1058.376,-74.102,-64.867,171.106,27.554,155.177
C07036=1058.383,-73.852,-64.878,171.107,27.556,155.177
C07037=1058.388,-73.602,-64.889,171.109,27.557,155.177
C07038=1058.394,-73.353,-64.901,171.111,27.559,155.178
C07039=1058.400,-73.103,-64.912,171.113,27.561,155.178
C07040=1058.407,-72.854,-64.924,171.115,27.563,155.178
C07041=1058.413,-72.604,-64.935,171.117,27.564,155.178
C07042=1058.418,-72.354,-64.947,171.119,27.565,155.178
C07043=1058.424,-72.105,-64.959,171.120,27.567,155.178
C07044=1058.431,-71.855,-64.970,171.122,27.569,155.178
C07045=1058.437,-71.606,-64.981,171.124,27.570,155.178
C07046=1058.442,-71.355,-64.993,171.126,27.571,155.178
C07047=1058.448,-71.106,-65.004,171.127,27.573,155.179
C07048=1058.455,-70.856,-65.016,171.129,27.575,155.179
C07049=1058.460,-70.607,-65.027,171.131,27.576,155.179
C07050=1058.467,-70.357,-65.039,171.132,27.578,155.179
C07051=1058.472,-70.107,-65.050,171.134,27.579,155.179
C07052=1058.479,-69.858,-65.062,171.136,27.581,155.179
C07053=1058.485,-69.608,-65.074,171.138,27.583,155.179
C07054=1058.491,-69.359,-65.085,171.139,27.584,155.179
C07055=1058.497,-69.108,-65.097,171.141,27.585,155.180
C07056=1058.503,-68.859,-65.109,171.143,27.587,155.180
C07057=1058.509,-68.609,-65.120,171.144,27.589,155.180
C07058=1058.515,-68.360,-65.131,171.147,27.591,155.180
C07059=1058.521,-68.110,-65.143,171.149,27.592,155.180
C07060=1058.527,-67.860,-65.155,171.151,27.594,155.180
C07061=1058.533,-67.611,-65.166,171.152,27.595,155.180
C07062=1058.540,-67.361,-65.178,171.154,27.597,155.180
C07063=1058.545,-67.112,-65.190,171.156,27.599,155.181
C07064=1058.552,-66.831,-65.203,171.157,27.600,155.181
C07065=1058.559,-66.550,-65.216,171.159,27.602,155.181
C07066=1058.565,-66.270,-65.229,171.162,27.604,155.181
C07067=1058.573,-65.989,-65.242,171.163,27.606,155.181
C07068=1058.579,-65.739,-65.254,171.165,27.607,155.181
C07069=1058.584,-65.489,-65.266,171.167,27.609,155.181
C07070=1058.591,-65.240,-65.278,171.169,27.611,155.181
C07071=1058.598,-64.990,-65.290,171.170,27.612,155.182
C07072=1058.603,-64.741,-65.301,171.172,27.614,155.182
C07073=1058.609,-64.491,-65.313,171.174,27.615,155.182
C07074=1058.616,-64.241,-65.325,171.176,27.617,155.182
C07075=1058.622,-63.992,-65.336,171.177,27.619,155.182
C07076=1058.628,-63.742,-65.348,171.179,27.620,155.182
C07077=1058.634,-63.492,-65.360,171.181,27.622,155.182
C07078=1058.640,-63.243,-65.371,171.183,27.624,155.182
C07079=1058.646,-62.993,-65.384,171.185,27.626,155.183
C07080=1058.652,-62.744,-65.396,171.187,27.627,155.183
C07081=1058.658,-62.494,-65.407,171.188,27.629,155.183
C07082=1058.664,-62.244,-65.419,171.190,27.631,155.183
C07083=1058.671,-61.995,-65.431,171.192,27.632,155.183
C07084=1058.677,-61.744,-65.442,171.194,27.633,155.183
C07085=1058.683,-61.496,-65.454,171.195,27.635,155.183
C07086=1058.689,-61.246,-65.466,171.197,27.637,155.184
C07087=1058.696,-60.996,-65.478,171.199,27.638,155.184
C07088=1058.701,-60.747,-65.489,171.200,27.640,155.184
C07089=1058.707,-60.497,-65.502,171.202,27.642,155.184
C07090=1058.714,-60.247,-65.514,171.204,27.644,155.184
C07091=1058.721,-59.998,-65.526,171.206,27.645,155.184
C07092=1058.726,-59.748,-65.538,171.207,27.647,155.184
C07093=1058.732,-59.498,-65.549,171.209,27.649,155.185
C07094=1058.738,-59.248,-65.562,171.211,27.650,155.185
C07095=1058.745,-58.999,-65.574,171.212,27.652,155.185
C07096=1058.751,-58.750,-65.585,171.214,27.654,155.185
C07097=1058.757,-58.500,-65.598,171.216,27.655,155.185
C07098=1058.763,-58.250,-65.609,171.217,27.657,155.185
C07099=1058.770,-58.000,-65.621,171.219,27.659,155.185
C07100=1058.776,-57.750,-65.634,171.221,27.660,155.186
C07101=1058.782,-57.501,-65.645,171.223,27.662,155.186
C07102=1058.788,-57.252,-65.657,171.225,27.664,155.186
C07103=1058.794,-57.002,-65.670,171.227,27.666,155.186
C07104=1058.801,-56.752,-65.682,171.229,27.667,155.186
C07105=1058.807,-56.502,-65.693,171.230,27.669,155.186
C07106=1058.813,-56.252,-65.705,171.232,27.671,155.186
C07107=1058.819,-56.003,-65.717,171.234,27.672,155.187
C07108=1058.825,-55.754,-65.730,171.235,27.674,155.187
C07109=1058.832,-55.504,-65.742,171.237,27.676,155.187
C07110=1058.838,-55.254,-65.754,171.239,27.677,155.187
C07111=1058.844,-55.005,-65.766,171.241,27.679,155.187
C07112=1058.851,-54.755,-65.778,171.242,27.681,155.187
C07113=1058.856,-54.506,-65.790,171.244,27.682,155.187
C07114=1058.863,-54.256,-65.802,171.246,27.684,155.188
C07115=1058.870,-54.007,-65.814,171.247,27.686,155.188
C07116=1058.876,-53.757,-65.827,171.249,27.688,155.188
C07117=1058.882,-53.507,-65.839,171.251,27.689,155.188
C07118=1058.888,-53.257,-65.851,171.253,27.691,155.188
C07119=1058.895,-53.008,-65.863,171.254,27.693,155.188
C07120=1058.901,-52.758,-65.875,171.256,27.694,155.188
C07121=1058.907,-52.509,-65.887,171.258,27.697,155.189
C07122=1058.913,-52.259,-65.899,171.259,27.698,155.189
C07123=1058.919,-52.010,-65.912,171.261,27.700,155.189
C07124=1058.926,-51.760,-65.924,171.263,27.702,155.189
C07125=1058.932,-51.510,-65.936,171.264,27.703,155.189
C07126=1058.938,-51.261,-65.948,171.266,27.705,155.189
C07127=1058.945,-51.011,-65.960,171.268,27.707,155.190
C07128=1058.952,-50.732,-65.974,171.270,27.709,155.190
C07129=1058.958,-50.452,-65.988,171.272,27.711,155.190
C07130=1058.966,-50.173,-66.002,171.274,27.713,155.190
C07131=1058.973,-49.894,-66.015,171.275,27.715,155.190
C07132=1058.979,-49.644,-66.028,171.277,27.716,155.190
C07133=1058.985,-49.394,-66.041,171.279,27.718,155.191
C07134=1058.991,-49.144,-66.053,171.280,27.720,155.191
C07135=1058.997,-48.895,-66.065,171.282,27.722,155.191
C07136=1059.003,-48.645,-66.077,171.284,27.724,155.191
C07137=1059.009,-48.396,-66.091,171.285,27.726,155.191
C07138=1059.015,-48.146,-66.103,171.287,27.728,155.192
C07139=1059.021,-47.897,-66.115,171.289,27.729,155.192
C07140=1059.027,-47.647,-66.128,171.291,27.732,155.192
C07141=1059.033,-47.397,-66.140,171.292,27.733,155.192
C07142=1059.040,-47.148,-66.153,171.294,27.735,155.192
C07143=1059.046,-46.898,-66.165,171.297,27.738,155.193
C07144=1059.052,-46.648,-66.178,171.298,27.739,155.193
C07145=1059.058,-46.398,-66.190,171.300,27.741,155.193
C07146=1059.064,-46.149,-66.202,171.302,27.743,155.193
C07147=1059.070,-45.900,-66.215,171.303,27.745,155.193
C07148=1059.076,-45.650,-66.228,171.305,27.747,155.193
C07149=1059.082,-45.400,-66.240,171.307,27.749,155.194
C07150=1059.089,-45.151,-66.252,171.308,27.750,155.194
C07151=1059.095,-44.902,-66.266,171.310,27.752,155.194
C07152=1059.101,-44.652,-66.278,171.312,27.754,155.194
C07153=1059.107,-44.402,-66.291,171.313,27.756,155.194
C07154=1059.113,-44.153,-66.304,171.315,27.758,155.195
C07155=1059.119,-43.903,-66.316,171.317,27.760,155.195
C07156=1059.125,-43.653,-66.329,171.318,27.762,155.195
C07157=1059.132,-43.404,-66.342,171.320,27.764,155.195
C07158=1059.137,-43.154,-66.354,171.322,27.766,155.195
C07159=1059.144,-42.904,-66.366,171.323,27.767,155.195
C07160=1059.150,-42.654,-66.379,171.325,27.770,155.196
C07161=1059.156,-42.405,-66.392,171.327,27.771,155.196
C07162=1059.162,-42.155,-66.405,171.328,27.774,155.196
C07163=1059.168,-41.906,-66.418,171.330,27.775,155.196
C07164=1059.175,-41.656,-66.430,171.332,27.777,155.196
C07165=1059.181,-41.407,-66.443,171.333,27.779,155.197
C07166=1059.187,-41.157,-66.456,171.335,27.781,155.197
C07167=1059.193,-40.907,-66.468,171.337,27.783,155.197
C07168=1059.199,-40.658,-66.481,171.338,27.785,155.197
C07169=1059.206,-40.409,-66.494,171.340,27.787,155.198
C07170=1059.212,-40.159,-66.506,171.342,27.789,155.198
C07171=1059.218,-39.909,-66.519,171.344,27.790,155.198
C07172=1059.224,-39.660,-66.532,171.345,27.793,155.198
C07173=1059.230,-39.410,-66.545,171.347,27.794,155.198
C07174=1059.236,-39.160,-66.558,171.348,27.797,155.198
C07175=1059.243,-38.911,-66.570,171.350,27.798,155.199
C07176=1059.249,-38.661,-66.583,171.352,27.801,155.199
C07177=1059.255,-38.411,-66.596,171.354,27.802,155.199
C07178=1059.262,-38.162,-66.609,171.354,27.804,155.199
C07179=1059.268,-37.912,-66.622,171.356,27.806,155.199
C07180=1059.274,-37.663,-66.635,171.358,27.808,155.200
C07181=1059.280,-37.413,-66.648,171.359,27.810,155.200
C07182=1059.286,-37.163,-66.661,171.361,27.812,155.200
C07183=1059.292,-36.914,-66.674,171.362,27.814,155.200
C07184=1059.298,-36.664,-66.687,171.364,27.816,155.201
C07185=1059.304,-36.415,-66.700,171.366,27.818,155.201
C07186=1059.310,-36.165,-66.712,171.368,27.820,155.201
C07187=1059.316,-35.916,-66.726,171.369,27.822,155.201
C07188=1059.322,-35.666,-66.738,171.371,27.825,155.202
C07189=1059.328,-35.417,-66.752,171.372,27.826,155.202
C07190=1059.334,-35.167,-66.765,171.374,27.828,155.202
C07191=1059.340,-34.917,-66.778,171.376,27.830,155.202
C07192=1059.347,-34.639,-66.793,171.377,27.832,155.202
C07193=1059.354,-34.359,-66.807,171.380,27.835,155.203
C07194=1059.361,-34.081,-66.822,171.382,27.837,155.203
C07195=1059.368,-33.802,-66.836,171.383,27.839,155.203
C07196=1059.374,-33.552,-66.849,171.385,27.842,155.203
C07197=1059.380,-33.303,-66.862,171.387,27.843,155.204
C07198=1059.386,-33.052,-66.876,171.388,27.846,155.204
C07199=1059.392,-32.803,-66.889,171.390,27.848,155.204
C07200=1059.398,-32.553,-66.902,171.392,27.850,155.204
C07201=1059.404,-32.304,-66.915,171.393,27.852,155.204
C07202=1059.411,-32.055,-66.928,171.395,27.853,155.205
C07203=1059.416,-31.805,-66.941,171.397,27.856,155.205
C07204=1059.423,-31.555,-66.954,171.398,27.858,155.205
C07205=1059.429,-31.305,-66.968,171.400,27.860,155.205
C07206=1059.436,-31.056,-66.981,171.402,27.862,155.206
C07207=1059.442,-30.806,-66.994,171.403,27.864,155.206
C07208=1059.448,-30.557,-67.007,171.405,27.866,155.206
C07209=1059.454,-30.308,-67.020,171.406,27.868,155.206
C07210=1059.459,-30.058,-67.033,171.408,27.870,155.207
C07211=1059.466,-29.808,-67.047,171.410,27.872,155.207
C07212=1059.472,-29.558,-67.060,171.411,27.874,155.207
C07213=1059.478,-29.309,-67.073,171.413,27.877,155.207
C07214=1059.485,-29.060,-67.087,171.415,27.878,155.207
C07215=1059.491,-28.810,-67.099,171.416,27.881,155.208
C07216=1059.497,-28.560,-67.113,171.417,27.883,155.208
C07217=1059.504,-28.311,-67.126,171.419,27.884,155.208
C07218=1059.510,-28.061,-67.139,171.420,27.886,155.208
C07219=1059.516,-27.812,-67.153,171.422,27.889,155.209
C07220=1059.521,-27.562,-67.166,171.424,27.890,155.209
C07221=1059.528,-27.312,-67.179,171.425,27.893,155.209
C07222=1059.534,-27.063,-67.193,171.427,27.895,155.209
C07223=1059.540,-26.814,-67.206,171.429,27.897,155.209
C07224=1059.547,-26.564,-67.219,171.430,27.899,155.210
C07225=1059.552,-26.315,-67.233,171.432,27.901,155.210
C07226=1059.559,-26.064,-67.246,171.434,27.903,155.210
C07227=1059.565,-25.815,-67.259,171.435,27.906,155.210
C07228=1059.570,-25.565,-67.273,171.437,27.907,155.211
C07229=1059.577,-25.316,-67.286,171.439,27.910,155.211
C07230=1059.583,-25.067,-67.300,171.440,27.912,155.211
C07231=1059.589,-24.816,-67.314,171.442,27.914,155.211
C07232=1059.595,-24.567,-67.327,171.444,27.916,155.212
C07233=1059.601,-24.318,-67.341,171.445,27.919,155.212
C07234=1059.607,-24.068,-67.354,171.447,27.920,155.212
C07235=1059.614,-23.818,-67.368,171.449,27.922,155.212
C07236=1059.620,-23.569,-67.381,171.450,27.925,155.213
C07237=1059.625,-23.320,-67.395,171.452,27.927,155.213
C07238=1059.631,-23.070,-67.408,171.452,27.929,155.213
C07239=1059.638,-22.820,-67.422,171.454,27.931,155.213
C07240=1059.644,-22.571,-67.436,171.456,27.933,155.214
C07241=1059.650,-22.321,-67.449,171.457,27.935,155.214
C07242=1059.656,-22.072,-67.462,171.459,27.937,155.214
C07243=1059.662,-21.822,-67.477,171.461,27.940,155.214
C07244=1059.668,-21.573,-67.490,171.462,27.942,155.215
C07245=1059.674,-21.323,-67.504,171.464,27.944,155.215
C07246=1059.680,-21.074,-67.517,171.466,27.946,155.215
C07247=1059.687,-20.824,-67.531,171.467,27.949,155.216
C07248=1059.692,-20.574,-67.545,171.469,27.950,155.216
C07249=1059.699,-20.325,-67.558,171.471,27.953,155.216
C07250=1059.705,-20.075,-67.571,171.472,27.955,155.216
C07251=1059.711,-19.826,-67.585,171.474,27.957,155.216
C07252=1059.717,-19.576,-67.599,171.475,27.959,155.217
C07253=1059.723,-19.326,-67.613,171.477,27.962,155.217
C07254=1059.729,-19.077,-67.626,171.479,27.964,155.217
C07255=1059.736,-18.827,-67.639,171.479,27.966,155.218
C07256=1059.742,-18.548,-67.655,171.482,27.968,155.218
C07257=1059.750,-18.268,-67.671,171.484,27.971,155.218
C07258=1059.757,-17.988,-67.686,171.485,27.973,155.218
